// TwinCAT 3 PLC project nott_ics
// ProgramVersion: 3.1.4024.0
// libraries:
//   CmpBitmapPool, * (System)
//   ESO LDC Comm Common Library, * (ESO)
//   ESO LDC Comm Tcp Library, * (ESO)
//   ESO LDC Common Library, * (ESO)
//   ESO LDC Cryo Library, * (ESO)
//   ESO LDC Motor Library, * (ESO)
//   ESO LDC Shutter Library, * (ESO)
//   ESO LDC Timer Library, * (ESO)
//   Tc2_EtherCAT, * (Beckhoff Automation GmbH)
//   Tc2_MC2, * (Beckhoff Automation GmbH)
//   Tc2_Standard, * (Beckhoff Automation GmbH)
//   Tc2_System, * (Beckhoff Automation GmbH)
//   Tc2_Utilities, * (Beckhoff Automation GmbH)
//   Tc3_Module, * (Beckhoff Automation GmbH)
//   VisuDialogs, * (System)
// project tree:
//   / CameraTrigs.TcTTO, GlobalTextList.TcGTLO, PlcTask.TcTTO, Visualization Manager.TcVMO (not stored), VISU_TASK.TcTTO
//   DUTs/Structures/ T_NOTT_STAT.TcDUT
//   DUTs/ T_NOTT_IR_CAMERA_DL_SYNC.TcDUT, T_NOTT_CAMERA_TIMESTAMPS_N_DL_POS.TcDUT
//   GVLs/ NOTT_GVL.TcGVL
//   HMI/DUTs/Subsystems/Tip_Tilt/ E_HMI_TIP_TILT_TABS.TcDUT
//   HMI/DUTs/System/ E_HMI_TABS.TcDUT
//   HMI/DUTs/Util/ E_HMI_COLORS.TcDUT, E_HMI_VOTER_TABS.TcDUT, T_ECAT_MODULE.TcDUT, T_HMI_COLORS.TcDUT
//   HMI/POUs/Devices/Cabinets/ FB_HMI_CABINETS.TcPOU
//   HMI/POUs/Devices/Control_Loops/ FB_HMI_CONTROL_LOOPS.TcPOU, FB_HMI_METIS_CTRL_TEMPERATURE.TcPOU
//   HMI/POUs/Devices/Control_Units/ FB_HMI_CONTROL_UNITS.TcPOU
//   HMI/POUs/Devices/Coolers/ FB_HMI_COOLERS.TcPOU
//   HMI/POUs/Devices/Detectors/ FB_HMI_DETECTORS.TcPOU
//   HMI/POUs/Devices/Heaters/ FB_HMI_HEATERS.TcPOU, FB_HMI_METIS_HEATER.TcPOU
//   HMI/POUs/Devices/Lakeshores/ FB_HMI_LAKESHORE.TcPOU
//   HMI/POUs/Devices/Pressures/ FB_HMI_PRESSURES.TcPOU
//   HMI/POUs/Devices/Pumps/ FB_HMI_PUMPS.TcPOU, FB_HMI_RP_BRANCH_A.TcPOU, FB_HMI_RP_BRANCH_B.TcPOU, FB_HMI_TP_BRANCH_A.TcPOU, FB_HMI_TP_BRANCH_B.TcPOU
//   HMI/POUs/Devices/RH/ FB_HMI_METIS_RH_SENSOR.TcPOU
//   HMI/POUs/Devices/Temperatures/Components/ FB_HMI_TEMP_VOTERS.TcPOU
//   HMI/POUs/Devices/Temperatures/ FB_HMI_TEMPERATURES.TcPOU
//   HMI/POUs/Devices/Valves/ FB_HMI_VALVES.TcPOU
//   HMI/POUs/Devices/Voters/ FB_HMI_VOTER.TcPOU
//   HMI/POUs/Events/ FB_HMI_EVENTS.TcPOU
//   HMI/POUs/CRYO_Interlocks/ FB_HMI_CRYO_INTERLOCKS.TcPOU
//   HMI/POUs/Services/ FB_HMI_SERVICES.TcPOU, FB_HMI_SERVICES_TIME.TcPOU
//   HMI/POUs/Services/Status/ FB_HMI_BUSY_STATUS.TcPOU, FB_HMI_HEALTH_STATUS.TcPOU, FB_HMI_STATUS.TcPOU, F_HMI_BUSY_TO_COLOR.TcPOU, F_HMI_HEALTH_BUSY_TO_COLOR.TcPOU, F_HMI_HEALTH_TO_COLOR.TcPOU
//   HMI/POUs/Subsystems/Beam_Splitter/ FB_HMI_CALIBRATION_BEAM_SPLITTER.TcPOU
//   HMI/POUs/Subsystems/Birefringence/ FB_HMI_BIREFRINGENCE.TcPOU
//   HMI/POUs/Subsystems/CO2_Pressure/ FB_HMI_CO2_PRESSURE_CONTROL.TcPOU
//   HMI/POUs/Subsystems/CO2_Translation_Stages/ FB_HMI_CO2_TRANS_STAGES.TcPOU
//   HMI/POUs/Subsystems/DelayLines/ FB_HMI_DELAY_LINES.TcPOU
//   HMI/POUs/Subsystems/Shutters/ FB_HMI_SHUTTERS.TcPOU
//   HMI/POUs/Subsystems/TipTilt/Components/ FB_HMI_TILT_A.TcPOU, FB_HMI_TILT_B.TcPOU, FB_HMI_TIP_A.TcPOU, FB_HMI_TIP_B.TcPOU
//   HMI/POUs/Subsystems/TipTilt/ FB_HMI_TIP_TILT.TcPOU
//   HMI/POUs/Subsystems/ZnSe_Actuators/ FB_HMI_ZNSE_ACTUATORS.TcPOU
//   HMI/POUs/Util/Button/ FB_HMI_BUTTON.TcPOU
//   HMI/POUs/Util/Component/ FB_HMI_COMPONENT.TcPOU
//   HMI/POUs/Util/Functions/ F_GetConnectionColor.TcPOU, F_GetConnectionString.TcPOU
//   HMI/ PRG_HMI.TcPOU, VISU_HMI.TcVIS
//   HMI/VISUs/Events/ VISU_HMI_EVENTS.TcVIS
//   HMI/VISUs/Home/ VISU_HMI_HOME.TcVIS
//   HMI/VISUs/ICS_Interlocks/ VISU_HMI_CRYO_INTERLOCKS.TcVIS
//   HMI/VISUs/Services/ VISU_HMI_SERVICES.TcVIS, VISU_HMI_SERVICES_TIME.TcVIS
//   HMI/VISUs/Subsystems/Beam_Splitter/ VISU_HMI_BEAM_SPLITTER.TcVIS
//   HMI/VISUs/Subsystems/Birefringence/ VISU_HMI_BIREFRINGENCE.TcVIS
//   HMI/VISUs/Subsystems/CO2_Pressure/ VISU_HMI_CO2_PRESSURE.TcVIS
//   HMI/VISUs/Subsystems/CO2_Translation_Stages/ VISU_HMI_CO2_TRANS_STAGES.TcVIS
//   HMI/VISUs/Subsystems/DelayLines/ VISU_HMI_DELAY_LINES.TcVIS
//   HMI/VISUs/Subsystems/Shutters/ VISU_HMI_SHUTTERS.TcVIS
//   HMI/VISUs/Subsystems/TipTilt/Components/ VISU_HMI_TILT_A.TcVIS, VISU_HMI_TILT_B.TcVIS, VISU_HMI_TIP_A.TcVIS, VISU_HMI_TIP_B.TcVIS
//   HMI/VISUs/Subsystems/TipTilt/ VISU_HMI_TIP_TILT.TcVIS
//   HMI/VISUs/Subsystems/ZnSe_Actuators/ VISU_HMI_ZNSE_ACTUATORS.TcVIS
//   HMI/VISUs/Templates/CO2_Valve/ GUI_TEMPLATE_ACTUATOR_ENG.TcVIS
//   HMI/VISUs/Templates/Motors/ GUI_TEMPLATE_MOTOR.TcVIS, GUI_TEMPLATE_NOTT_MOTOR_CONFIG.TcVIS, GUI_TEMPLATE_NOTT_MOTOR_CONTROL.TcVIS
//   HMI/VISUs/Templates/ NOTT_Images.TcIPO (not stored)
//   HMI/VISUs/Templates/Shutters/ GUI_TEMPLATE_NOTT_SHUTTER.TcVIS, GUI_TEMPLATE_SHUTTER_CONTROL.TcVIS
//   HMI/VISUs/Util/Button/ VISU_HMI_BUTTON_IMAGES.TcIPO (not stored), VISU_HMI_ROUTINES_BUTTON.TcVIS, VISU_HMI_SUBSUBSYSTEM_BUTTON.TcVIS, VISU_HMI_SUBSYSTEM_BUTTON.TcVIS, VISU_HMI_SYSTEM_BUTTON.TcVIS
//   HMI/VISUs/Util/ ICONS_IMAGE_POOL.TcIPO (not stored)
//   POUs/Camera_Triggers/ INFRATEC_TRIGERS.TcPOU
//   POUs/Cryo_Interlocks/ FB_NOTT_CRYO_INTERLOCKS.TcPOU
//   POUs/Devices/NOTT_Motor/ FB_NOTT_MOTOR.TcPOU
//   POUs/EVENTS/ FB_NOTT_EVENTS.TcPOU
//   POUs/Functions/ F_SysTimeToString.TcPOU
//   POUs/ MAIN.TcPOU
//   POUs/Services/ FB_SERVICES.TcPOU
//   POUs/Subsystems/ FB_NOTT_CO2_PRESSURE_CONTROL.TcPOU, FB_NOTT_CALIBRATION_BEAM_SPLITTER.TcPOU, FB_NOTT_ZNSE_ACTUATORS.TcPOU, FB_NOTT_DELAY_LINES.TcPOU, FB_NOTT_SHUTTERS.TcPOU, FB_NOTT_CO2_TRANS_STAGES.TcPOU, FB_NOTT_TIP_TILT.TcPOU, FB_NOTT_BIREFRINGENCE.TcPOU
//   POUs/System/ FB_NOTT_CRYO_CTRL.TcPOU, FB_NOTT_ICS.TcPOU
//   POUs/Valve/ FB_CRYO_BIN_CTRL.TcPOU, FB_CRYO_VALVE_CTRL.TcPOU
//   VISUs/GUIs/Cryo/ GUI_CRYO_TEMPS.TcVIS
//   VISUs/GUIs/NBS/ GUI_NOTT_NBS.TcVIS
//   VISUs/GUIs/Shutters/ GUI_TEST_STEPPER_SHUTTER.TcVIS, GUI_NOTT_SHUTTERS.TcVIS
//   VISUs/GUIs/Templates/ TEMPLATE_NOTT_CRYO_TEMPS.TcVIS
//   VISUs/GUIs/Delay_Lines/ GUI_NOTT_DL_CONFIG.TcVIS, GUI_NOTT_DL_CTRL.TcVIS
//   VISUs/GUIs/ GUI_NOTT_DL_1.TcVIS
//   VISUs/GUIs/Time/ GUI_NOTT_TIME.TcVIS
//   VISUs/GUIs/TipTilt/ GUI_NOTT_TIP_A_CONFIG.TcVIS, GUI_NOTT_TIP_B_CONFIG.TcVIS, GUI_NOTT_TILT_B_CONFIG.TcVIS, GUI_NOTT_TILT_A_CONFIG.TcVIS, GUI_NOTT_TIP_A_CTRL.TcVIS, GUI_NOTT_TIP_B_CTRL.TcVIS, GUI_NOTT_TILT_A_CTRL.TcVIS, GUI_NOTT_TILT_B_CTRL.TcVIS
//   VISUs/Templates/ MOTOR_CONTROL.TcVIS
// real-time tasks:
//   TASK PlcTask: cycle T#10ms, priority 20, ADS port 350
//   TASK CameraTrigs: cycle T#1ms, priority 1, ADS port 351
//   TASK VISU_TASK: cycle T#200000us, priority 30, ADS port 352
// motion (NC):
//   TASK NC-Task 1 SAF: cycle T#2ms, priority 4, ADS port 501
//   TASK NC-Task 1 SVB: cycle T#10ms, priority 8, ADS port 511
//   AXIS NTPA1 (id 23)
//     Dynamic: AccelerationMaximum=1.8, DecelerationMaximum=1.8, Acceleration=0.2525, Deceleration=0.2525, Jerk=15.9390625
//     Velo: RefSearch=0.05, RefSync=0.05, SlowManual=0.05, FastManual=0.1, Fast=0.4, Maximum=0.4
//     OtherSettings: AllowMotionCmdToSlave=true, PulseDistancePos=0.05, PulseDistanceNeg=0.05
//     encoder EncType=4
//       EncPara: ScaleFactorNumerator=3.05e-05, MaxCount=#x0000ffff
//         Inc: RefSoftSyncMask=#x0000ffff
//     drive DrvType=23
//       Analog: VeloReferenz=0.4, TorqueSetpointScale=10, ScaleFactorActTorque=0.1
//       TimeComp: TaskDelayCycles=1
//     controller CtrType=13
//       CtrPara: PriorControlFactor=1
//         PID: PosKp=50, PosTn=5, PosTd=0.5, DeadBandPosition=1e-05
//         Observer: ObserverMode=1, MotorTorqueConstant=2, BandWidth=20
//   AXIS NTPA2 (id 24)
//     Dynamic: AccelerationMaximum=1.8, DecelerationMaximum=1.8, Acceleration=0.2525, Deceleration=0.2525, Jerk=15.9390625
//     Velo: RefSearch=0.05, RefSync=0.05, SlowManual=0.05, FastManual=0.1, Fast=0.4, Maximum=0.4
//     OtherSettings: AllowMotionCmdToSlave=true, PulseDistancePos=0.05, PulseDistanceNeg=0.05
//     encoder EncType=4
//       EncPara: ScaleFactorNumerator=3.05e-05, MaxCount=#x0000ffff
//         Inc: RefSoftSyncMask=#x0000ffff
//     drive DrvType=23
//       Analog: VeloReferenz=0.4, TorqueSetpointScale=10, ScaleFactorActTorque=0.1
//       TimeComp: TaskDelayCycles=1
//     controller CtrType=13
//       CtrPara: PriorControlFactor=1
//         PID: PosKp=50, PosTn=5, PosTd=0.5, DeadBandPosition=1e-05
//         Observer: ObserverMode=1, MotorTorqueConstant=2, BandWidth=20
//   AXIS NTPA3 (id 25)
//     Dynamic: AccelerationMaximum=1.8, DecelerationMaximum=1.8, Acceleration=0.2525, Deceleration=0.2525, Jerk=15.9390625
//     Velo: RefSearch=0.05, RefSync=0.05, SlowManual=0.05, FastManual=0.1, Fast=0.4, Maximum=0.4
//     OtherSettings: AllowMotionCmdToSlave=true, PulseDistancePos=0.05, PulseDistanceNeg=0.05
//     encoder EncType=4
//       EncPara: ScaleFactorNumerator=3.05e-05, MaxCount=#x0000ffff
//         Inc: RefSoftSyncMask=#x0000ffff
//     drive DrvType=23
//       Analog: VeloReferenz=0.4, TorqueSetpointScale=10, ScaleFactorActTorque=0.1
//       TimeComp: TaskDelayCycles=1
//     controller CtrType=13
//       CtrPara: PriorControlFactor=1
//         PID: PosKp=50, PosTn=5, PosTd=0.5, DeadBandPosition=1e-05
//         Observer: ObserverMode=1, MotorTorqueConstant=2, BandWidth=20
//   AXIS NTPA4 (id 26)
//     Dynamic: AccelerationMaximum=1.8, DecelerationMaximum=1.8, Acceleration=0.2525, Deceleration=0.2525, Jerk=15.9390625
//     Velo: RefSearch=0.05, RefSync=0.05, SlowManual=0.05, FastManual=0.1, Fast=0.4, Maximum=0.4
//     OtherSettings: AllowMotionCmdToSlave=true, PulseDistancePos=0.05, PulseDistanceNeg=0.05
//     encoder EncType=4
//       EncPara: ScaleFactorNumerator=3.05e-05, MaxCount=#x0000ffff
//         Inc: RefSoftSyncMask=#x0000ffff
//     drive DrvType=23
//       Analog: VeloReferenz=0.4, TorqueSetpointScale=10, ScaleFactorActTorque=0.1
//       TimeComp: TaskDelayCycles=1
//     controller CtrType=13
//       CtrPara: PriorControlFactor=1
//         PID: PosKp=50, PosTn=5, PosTd=0.5, DeadBandPosition=1e-05
//         Observer: ObserverMode=1, MotorTorqueConstant=2, BandWidth=20
//   AXIS NTTA1 (id 27)
//     Dynamic: AccelerationMaximum=1.8, DecelerationMaximum=1.8, Acceleration=0.2525, Deceleration=0.2525, Jerk=15.9390625
//     Velo: RefSearch=0.05, RefSync=0.05, SlowManual=0.05, FastManual=0.1, Fast=0.4, Maximum=0.4
//     OtherSettings: AllowMotionCmdToSlave=true, PulseDistancePos=0.05, PulseDistanceNeg=0.05
//     encoder EncType=4
//       EncPara: ScaleFactorNumerator=3.05e-05, MaxCount=#x0000ffff
//         Inc: RefSoftSyncMask=#x0000ffff
//     drive DrvType=23
//       Analog: VeloReferenz=0.4, TorqueSetpointScale=10, ScaleFactorActTorque=0.1
//       TimeComp: TaskDelayCycles=1
//     controller CtrType=13
//       CtrPara: PriorControlFactor=1
//         PID: PosKp=50, PosTn=5, PosTd=0.5, DeadBandPosition=1e-05
//         Observer: ObserverMode=1, MotorTorqueConstant=2, BandWidth=20
//   AXIS NTTA2 (id 28)
//     Dynamic: AccelerationMaximum=1.8, DecelerationMaximum=1.8, Acceleration=0.2525, Deceleration=0.2525, Jerk=15.9390625
//     Velo: RefSearch=0.05, RefSync=0.05, SlowManual=0.05, FastManual=0.1, Fast=0.4, Maximum=0.4
//     OtherSettings: AllowMotionCmdToSlave=true, PulseDistancePos=0.05, PulseDistanceNeg=0.05
//     encoder EncType=4
//       EncPara: ScaleFactorNumerator=3.05e-05, MaxCount=#x0000ffff
//         Inc: RefSoftSyncMask=#x0000ffff
//     drive DrvType=23
//       Analog: VeloReferenz=0.4, TorqueSetpointScale=10, ScaleFactorActTorque=0.1
//       TimeComp: TaskDelayCycles=1
//     controller CtrType=13
//       CtrPara: PriorControlFactor=1
//         PID: PosKp=50, PosTn=5, PosTd=0.5, DeadBandPosition=1e-05
//         Observer: ObserverMode=1, MotorTorqueConstant=2, BandWidth=20
//   AXIS NTTA3 (id 29)
//     Dynamic: AccelerationMaximum=1.8, DecelerationMaximum=1.8, Acceleration=0.2525, Deceleration=0.2525, Jerk=15.9390625
//     Velo: RefSearch=0.05, RefSync=0.05, SlowManual=0.05, FastManual=0.1, Fast=0.4, Maximum=0.4
//     OtherSettings: AllowMotionCmdToSlave=true, PulseDistancePos=0.05, PulseDistanceNeg=0.05
//     encoder EncType=4
//       EncPara: ScaleFactorNumerator=3.05e-05, MaxCount=#x0000ffff
//         Inc: RefSoftSyncMask=#x0000ffff
//     drive DrvType=23
//       Analog: VeloReferenz=0.4, TorqueSetpointScale=10, ScaleFactorActTorque=0.1
//       TimeComp: TaskDelayCycles=1
//     controller CtrType=13
//       CtrPara: PriorControlFactor=1
//         PID: PosKp=50, PosTn=5, PosTd=0.5, DeadBandPosition=1e-05
//         Observer: ObserverMode=1, MotorTorqueConstant=2, BandWidth=20
//   AXIS NTTA4 (id 30)
//     Dynamic: AccelerationMaximum=1.8, DecelerationMaximum=1.8, Acceleration=0.2525, Deceleration=0.2525, Jerk=15.9390625
//     Velo: RefSearch=0.05, RefSync=0.05, SlowManual=0.05, FastManual=0.1, Fast=0.4, Maximum=0.4
//     OtherSettings: AllowMotionCmdToSlave=true, PulseDistancePos=0.05, PulseDistanceNeg=0.05
//     encoder EncType=4
//       EncPara: ScaleFactorNumerator=3.05e-05, MaxCount=#x0000ffff
//         Inc: RefSoftSyncMask=#x0000ffff
//     drive DrvType=23
//       Analog: VeloReferenz=0.4, TorqueSetpointScale=10, ScaleFactorActTorque=0.1
//       TimeComp: TaskDelayCycles=1
//     controller CtrType=13
//       CtrPara: PriorControlFactor=1
//         PID: PosKp=50, PosTn=5, PosTd=0.5, DeadBandPosition=1e-05
//         Observer: ObserverMode=1, MotorTorqueConstant=2, BandWidth=20
//   AXIS NTPB1 (id 31)
//     Dynamic: AccelerationMaximum=1.8, DecelerationMaximum=1.8, Acceleration=0.2525, Deceleration=0.2525, Jerk=15.9390625
//     Velo: RefSearch=0.05, RefSync=0.05, SlowManual=0.05, FastManual=0.1, Fast=0.4, Maximum=0.4
//     OtherSettings: AllowMotionCmdToSlave=true, PulseDistancePos=0.05, PulseDistanceNeg=0.05
//     encoder EncType=4
//       EncPara: ScaleFactorNumerator=3.05e-05, MaxCount=#x0000ffff
//         Inc: RefSoftSyncMask=#x0000ffff
//     drive DrvType=23
//       Analog: VeloReferenz=0.4, TorqueSetpointScale=10, ScaleFactorActTorque=0.1
//       TimeComp: TaskDelayCycles=1
//     controller CtrType=13
//       CtrPara: PriorControlFactor=1
//         PID: PosKp=50, PosTn=5, PosTd=0.5, DeadBandPosition=1e-05
//         Observer: ObserverMode=1, MotorTorqueConstant=2, BandWidth=20
//   AXIS NTPB2 (id 32)
//     Dynamic: AccelerationMaximum=1.8, DecelerationMaximum=1.8, Acceleration=0.2525, Deceleration=0.2525, Jerk=15.9390625
//     Velo: RefSearch=0.05, RefSync=0.05, SlowManual=0.05, FastManual=0.1, Fast=0.4, Maximum=0.4
//     OtherSettings: AllowMotionCmdToSlave=true, PulseDistancePos=0.05, PulseDistanceNeg=0.05
//     encoder EncType=4
//       EncPara: ScaleFactorNumerator=3.05e-05, MaxCount=#x0000ffff
//         Inc: RefSoftSyncMask=#x0000ffff
//     drive DrvType=23
//       Analog: VeloReferenz=0.4, TorqueSetpointScale=10, ScaleFactorActTorque=0.1
//       TimeComp: TaskDelayCycles=1
//     controller CtrType=13
//       CtrPara: PriorControlFactor=1
//         PID: PosKp=50, PosTn=5, PosTd=0.5, DeadBandPosition=1e-05
//         Observer: ObserverMode=1, MotorTorqueConstant=2, BandWidth=20
//   AXIS NTPB3 (id 33)
//     Dynamic: AccelerationMaximum=1.8, DecelerationMaximum=1.8, Acceleration=0.2525, Deceleration=0.2525, Jerk=15.9390625
//     Velo: RefSearch=0.05, RefSync=0.05, SlowManual=0.05, FastManual=0.1, Fast=0.4, Maximum=0.4
//     OtherSettings: AllowMotionCmdToSlave=true, PulseDistancePos=0.05, PulseDistanceNeg=0.05
//     encoder EncType=4
//       EncPara: ScaleFactorNumerator=3.05e-05, MaxCount=#x0000ffff
//         Inc: RefSoftSyncMask=#x0000ffff
//     drive DrvType=23
//       Analog: VeloReferenz=0.4, TorqueSetpointScale=10, ScaleFactorActTorque=0.1
//       TimeComp: TaskDelayCycles=1
//     controller CtrType=13
//       CtrPara: PriorControlFactor=1
//         PID: PosKp=50, PosTn=5, PosTd=0.5, DeadBandPosition=1e-05
//         Observer: ObserverMode=1, MotorTorqueConstant=2, BandWidth=20
//   AXIS NTPB4 (id 34)
//     Dynamic: AccelerationMaximum=1.8, DecelerationMaximum=1.8, Acceleration=0.2525, Deceleration=0.2525, Jerk=15.9390625
//     Velo: RefSearch=0.05, RefSync=0.05, SlowManual=0.05, FastManual=0.1, Fast=0.4, Maximum=0.4
//     OtherSettings: AllowMotionCmdToSlave=true, PulseDistancePos=0.05, PulseDistanceNeg=0.05
//     encoder EncType=4
//       EncPara: ScaleFactorNumerator=3.05e-05, MaxCount=#x0000ffff
//         Inc: RefSoftSyncMask=#x0000ffff
//     drive DrvType=23
//       Analog: VeloReferenz=0.4, TorqueSetpointScale=10, ScaleFactorActTorque=0.1
//       TimeComp: TaskDelayCycles=1
//     controller CtrType=13
//       CtrPara: PriorControlFactor=1
//         PID: PosKp=50, PosTn=5, PosTd=0.5, DeadBandPosition=1e-05
//         Observer: ObserverMode=1, MotorTorqueConstant=2, BandWidth=20
//   AXIS NTTB1 (id 36)
//     Dynamic: AccelerationMaximum=1.8, DecelerationMaximum=1.8, Acceleration=0.2525, Deceleration=0.2525, Jerk=15.9390625
//     Velo: RefSearch=0.05, RefSync=0.05, SlowManual=0.05, FastManual=0.1, Fast=0.4, Maximum=0.4
//     OtherSettings: AllowMotionCmdToSlave=true, PulseDistancePos=0.05, PulseDistanceNeg=0.05
//     encoder EncType=4
//       EncPara: ScaleFactorNumerator=3.05e-05, MaxCount=#x0000ffff
//         Inc: RefSoftSyncMask=#x0000ffff
//     drive DrvType=23
//       Analog: VeloReferenz=0.4, TorqueSetpointScale=10, ScaleFactorActTorque=0.1
//       TimeComp: TaskDelayCycles=1
//     controller CtrType=13
//       CtrPara: PriorControlFactor=1
//         PID: PosKp=50, PosTn=5, PosTd=0.5, DeadBandPosition=1e-05
//         Observer: ObserverMode=1, MotorTorqueConstant=2, BandWidth=20
//   AXIS NTTB2 (id 37)
//     Dynamic: AccelerationMaximum=1.8, DecelerationMaximum=1.8, Acceleration=0.2525, Deceleration=0.2525, Jerk=15.9390625
//     Velo: RefSearch=0.05, RefSync=0.05, SlowManual=0.05, FastManual=0.1, Fast=0.4, Maximum=0.4
//     OtherSettings: AllowMotionCmdToSlave=true, PulseDistancePos=0.05, PulseDistanceNeg=0.05
//     encoder EncType=4
//       EncPara: ScaleFactorNumerator=3.05e-05, MaxCount=#x0000ffff
//         Inc: RefSoftSyncMask=#x0000ffff
//     drive DrvType=23
//       Analog: VeloReferenz=0.4, TorqueSetpointScale=10, ScaleFactorActTorque=0.1
//       TimeComp: TaskDelayCycles=1
//     controller CtrType=13
//       CtrPara: PriorControlFactor=1
//         PID: PosKp=50, PosTn=5, PosTd=0.5, DeadBandPosition=1e-05
//         Observer: ObserverMode=1, MotorTorqueConstant=2, BandWidth=20
//   AXIS NTTB3 (id 38)
//     Dynamic: AccelerationMaximum=1.8, DecelerationMaximum=1.8, Acceleration=0.2525, Deceleration=0.2525, Jerk=15.9390625
//     Velo: RefSearch=0.05, RefSync=0.05, SlowManual=0.05, FastManual=0.1, Fast=0.4, Maximum=0.4
//     OtherSettings: AllowMotionCmdToSlave=true, PulseDistancePos=0.05, PulseDistanceNeg=0.05
//     encoder EncType=4
//       EncPara: ScaleFactorNumerator=3.05e-05, MaxCount=#x0000ffff
//         Inc: RefSoftSyncMask=#x0000ffff
//     drive DrvType=23
//       Analog: VeloReferenz=0.4, TorqueSetpointScale=10, ScaleFactorActTorque=0.1
//       TimeComp: TaskDelayCycles=1
//     controller CtrType=13
//       CtrPara: PriorControlFactor=1
//         PID: PosKp=50, PosTn=5, PosTd=0.5, DeadBandPosition=1e-05
//         Observer: ObserverMode=1, MotorTorqueConstant=2, BandWidth=20
//   AXIS NTTB4 (id 39)
//     Dynamic: AccelerationMaximum=1.8, DecelerationMaximum=1.8, Acceleration=0.2525, Deceleration=0.2525, Jerk=15.9390625
//     Velo: RefSearch=0.05, RefSync=0.05, SlowManual=0.05, FastManual=0.1, Fast=0.4, Maximum=0.4
//     OtherSettings: AllowMotionCmdToSlave=true, PulseDistancePos=0.05, PulseDistanceNeg=0.05
//     encoder EncType=4
//       EncPara: ScaleFactorNumerator=3.05e-05, MaxCount=#x0000ffff
//         Inc: RefSoftSyncMask=#x0000ffff
//     drive DrvType=23
//       Analog: VeloReferenz=0.4, TorqueSetpointScale=10, ScaleFactorActTorque=0.1
//       TimeComp: TaskDelayCycles=1
//     controller CtrType=13
//       CtrPara: PriorControlFactor=1
//         PID: PosKp=50, PosTn=5, PosTd=0.5, DeadBandPosition=1e-05
//         Observer: ObserverMode=1, MotorTorqueConstant=2, BandWidth=20
//   AXIS NDL1 (id 19)
//     Dynamic: AccelerationMaximum=0.3, DecelerationMaximum=0.3, Acceleration=0.3, Deceleration=0.3, Jerk=0.5
//     Velo: RefSearch=0.05, RefSync=0.05, SlowManual=0.02, FastManual=0.075, Fast=0.2, Maximum=0.2
//     OtherSettings: AllowMotionCmdToSlave=true, PulseDistancePos=0.02, PulseDistanceNeg=0.02
//     encoder EncType=4
//       EncPara: ScaleFactorNumerator=1.5259e-06, MaxCount=#x0000ffff
//         Inc: RefSoftSyncMask=#x0000ffff
//     drive DrvType=24
//       Analog: VeloReferenz=0.2, TorqueSetpointScale=10, ScaleFactorActTorque=0.1
//       TimeComp: TaskDelayCycles=1
//     controller CtrType=1
//       CtrPara: PriorControlFactor=1
//         Observer: BandWidth=20
//   AXIS NDL2 (id 20)
//     Dynamic: AccelerationMaximum=0.3, DecelerationMaximum=0.3, Acceleration=0.3, Deceleration=0.3, Jerk=0.5
//     Velo: RefSearch=0.05, RefSync=0.05, SlowManual=0.02, FastManual=0.075, Fast=0.2, Maximum=0.2
//     OtherSettings: AllowMotionCmdToSlave=true, PulseDistancePos=0.02, PulseDistanceNeg=0.02
//     encoder EncType=4
//       EncPara: ScaleFactorNumerator=1.5259e-06, MaxCount=#x0000ffff
//         Inc: RefSoftSyncMask=#x0000ffff
//     drive DrvType=24
//       Analog: VeloReferenz=0.2, TorqueSetpointScale=10, ScaleFactorActTorque=0.1
//       TimeComp: TaskDelayCycles=1
//     controller CtrType=1
//       CtrPara: PriorControlFactor=1
//         Observer: BandWidth=20
//   AXIS NDL3 (id 21)
//     Dynamic: AccelerationMaximum=0.3, DecelerationMaximum=0.3, Acceleration=0.3, Deceleration=0.3, Jerk=0.5
//     Velo: RefSearch=0.05, RefSync=0.05, SlowManual=0.02, FastManual=0.075, Fast=0.2, Maximum=0.2
//     OtherSettings: AllowMotionCmdToSlave=true, PulseDistancePos=0.02, PulseDistanceNeg=0.02
//     encoder EncType=4
//       EncPara: ScaleFactorNumerator=1.5259e-06, MaxCount=#x0000ffff
//         Inc: RefSoftSyncMask=#x0000ffff
//     drive DrvType=24
//       Analog: VeloReferenz=0.2, TorqueSetpointScale=10, ScaleFactorActTorque=0.1
//       TimeComp: TaskDelayCycles=1
//     controller CtrType=1
//       CtrPara: PriorControlFactor=1
//         Observer: BandWidth=20
//   AXIS NDL4 (id 22)
//     Dynamic: AccelerationMaximum=0.3, DecelerationMaximum=0.3, Acceleration=0.3, Deceleration=0.3, Jerk=0.5
//     Velo: RefSearch=0.05, RefSync=0.05, SlowManual=0.02, FastManual=0.075, Fast=0.2, Maximum=0.2
//     OtherSettings: AllowMotionCmdToSlave=true, PulseDistancePos=0.02, PulseDistanceNeg=0.02
//     encoder EncType=4
//       EncPara: ScaleFactorNumerator=1.5259e-06, MaxCount=#x0000ffff
//         Inc: RefSoftSyncMask=#x0000ffff
//     drive DrvType=24
//       Analog: VeloReferenz=0.2, TorqueSetpointScale=10, ScaleFactorActTorque=0.1
//       TimeComp: TaskDelayCycles=1
//     controller CtrType=1
//       CtrPara: PriorControlFactor=1
//         Observer: BandWidth=20
//   AXIS NSH1 (id 35)
//     Dynamic: AccelerationMaximum=100, DecelerationMaximum=100, Acceleration=9, Deceleration=9, Jerk=1000
//     Velo: RefSearch=3, RefSync=3, SlowManual=3, FastManual=5, Fast=30, Maximum=35
//     PositionAreaControl: Enable=false
//     OtherSettings: AllowMotionCmdToSlave=true, PulseDistancePos=1, PulseDistanceNeg=1
//     encoder EncType=4
//       EncPara: ScaleFactorNumerator=0.00234375, MaxCount=#x0000ffff
//         Inc: RefSoftSyncMask=#x0000ffff
//     drive DrvType=24
//       Analog: VeloReferenz=35, TorqueSetpointScale=10, ScaleFactorActTorque=0.1
//       TimeComp: TaskDelayCycles=1
//     controller CtrType=1
//       CtrPara: PriorControlFactor=1
//         PosDiffControl: Enable=false
//         PID: PosKp=10
//         Observer: BandWidth=20
//   AXIS NSH2 (id 16)
//     Dynamic: AccelerationMaximum=100, DecelerationMaximum=100, Acceleration=9, Deceleration=9, Jerk=1000
//     Velo: RefSearch=3, RefSync=3, SlowManual=3, FastManual=5, Fast=30, Maximum=35
//     PositionAreaControl: Enable=false
//     OtherSettings: AllowMotionCmdToSlave=true, PulseDistancePos=1, PulseDistanceNeg=1
//     encoder EncType=4
//       EncPara: ScaleFactorNumerator=0.00234375, MaxCount=#x0000ffff
//         Inc: RefSoftSyncMask=#x0000ffff
//     drive DrvType=24
//       Analog: VeloReferenz=35, TorqueSetpointScale=10, ScaleFactorActTorque=0.1
//       TimeComp: TaskDelayCycles=1
//     controller CtrType=1
//       CtrPara: PriorControlFactor=1
//         PosDiffControl: Enable=false
//         PID: PosKp=10
//         Observer: BandWidth=20
//   AXIS NSH3 (id 17)
//     Dynamic: AccelerationMaximum=100, DecelerationMaximum=100, Acceleration=9, Deceleration=9, Jerk=1000
//     Velo: RefSearch=3, RefSync=3, SlowManual=3, FastManual=5, Fast=30, Maximum=35
//     PositionAreaControl: Enable=false
//     OtherSettings: AllowMotionCmdToSlave=true, PulseDistancePos=1, PulseDistanceNeg=1
//     encoder EncType=4
//       EncPara: ScaleFactorNumerator=0.00234375, MaxCount=#x0000ffff
//         Inc: RefSoftSyncMask=#x0000ffff
//     drive DrvType=24
//       Analog: VeloReferenz=35, TorqueSetpointScale=10, ScaleFactorActTorque=0.1
//       TimeComp: TaskDelayCycles=1
//     controller CtrType=1
//       CtrPara: PriorControlFactor=1
//         PosDiffControl: Enable=false
//         PID: PosKp=10
//         Observer: BandWidth=20
//   AXIS NSH4 (id 18)
//     Dynamic: AccelerationMaximum=200, DecelerationMaximum=200, Acceleration=9, Deceleration=9, Jerk=726.357
//     Velo: RefSearch=3, RefSync=3, SlowManual=3, FastManual=5, Fast=30, Maximum=35
//     PositionAreaControl: Enable=false
//     OtherSettings: AllowMotionCmdToSlave=true, PulseDistancePos=1, PulseDistanceNeg=1
//     encoder EncType=4
//       EncPara: ScaleFactorNumerator=0.00234375, MaxCount=#x0000ffff
//         Inc: RefSoftSyncMask=#x0000ffff
//     drive DrvType=24
//       Analog: VeloReferenz=35, TorqueSetpointScale=10, ScaleFactorActTorque=0.1
//       TimeComp: TaskDelayCycles=1
//     controller CtrType=1
//       CtrPara: PriorControlFactor=1
//         PosDiffControl: Enable=false
//         PID: PosKp=10
//         Observer: BandWidth=20
//   AXIS NCP1 (id 1)
//     Dynamic: AccelerationMaximum=4.5, DecelerationMaximum=4.5, Acceleration=4.5, Deceleration=4.5, Jerk=9
//     Velo: RefSearch=0.5, RefSync=0.5, SlowManual=0.05, FastManual=0.05, Fast=2, Maximum=2.3
//     OtherSettings: AllowMotionCmdToSlave=true, PulseDistancePos=0.02, PulseDistanceNeg=0.02
//     encoder EncType=4
//       EncPara: ScaleFactorNumerator=2.893937e-05, MaxCount=#x0000ffff
//         Inc: RefSoftSyncMask=#x0000ffff
//     drive DrvType=23
//       Analog: VeloReferenz=2.3, TorqueSetpointScale=10, ScaleFactorActTorque=0.1
//       TimeComp: TaskDelayCycles=1
//     controller CtrType=1
//       CtrPara: PriorControlFactor=1
//         Observer: BandWidth=20
//   AXIS NCP2 (id 2)
//     Dynamic: AccelerationMaximum=4.5, DecelerationMaximum=4.5, Acceleration=4.5, Deceleration=4.5, Jerk=9
//     Velo: RefSearch=0.5, RefSync=0.5, SlowManual=0.05, FastManual=0.05, Fast=2, Maximum=2.3
//     OtherSettings: AllowMotionCmdToSlave=true, PulseDistancePos=0.02, PulseDistanceNeg=0.02
//     encoder EncType=4
//       EncPara: ScaleFactorNumerator=2.893937e-05, MaxCount=#x0000ffff
//         Inc: RefSoftSyncMask=#x0000ffff
//     drive DrvType=23
//       Analog: VeloReferenz=2.3, TorqueSetpointScale=10, ScaleFactorActTorque=0.1
//       TimeComp: TaskDelayCycles=1
//     controller CtrType=1
//       CtrPara: PriorControlFactor=1
//         Observer: BandWidth=20
//   AXIS NCP3 (id 3)
//     Dynamic: AccelerationMaximum=4.5, DecelerationMaximum=4.5, Acceleration=4.5, Deceleration=4.5, Jerk=9
//     Velo: RefSearch=0.5, RefSync=0.5, SlowManual=0.05, FastManual=0.05, Fast=2, Maximum=2.3
//     OtherSettings: AllowMotionCmdToSlave=true, PulseDistancePos=0.02, PulseDistanceNeg=0.02
//     encoder EncType=4
//       EncPara: ScaleFactorNumerator=2.893937e-05, MaxCount=#x0000ffff
//         Inc: RefSoftSyncMask=#x0000ffff
//     drive DrvType=23
//       Analog: VeloReferenz=2.3, TorqueSetpointScale=10, ScaleFactorActTorque=0.1
//       TimeComp: TaskDelayCycles=1
//     controller CtrType=1
//       CtrPara: PriorControlFactor=1
//         Observer: BandWidth=20
//   AXIS NCP4 (id 4)
//     Dynamic: AccelerationMaximum=4.5, DecelerationMaximum=4.5, Acceleration=4.5, Deceleration=4.5, Jerk=9
//     Velo: RefSearch=0.5, RefSync=0.5, SlowManual=0.05, FastManual=0.05, Fast=2, Maximum=2.3
//     OtherSettings: AllowMotionCmdToSlave=true, PulseDistancePos=0.02, PulseDistanceNeg=0.02
//     encoder EncType=4
//       EncPara: ScaleFactorNumerator=2.893937e-05, MaxCount=#x0000ffff
//         Inc: RefSoftSyncMask=#x0000ffff
//     drive DrvType=23
//       Analog: VeloReferenz=2.3, TorqueSetpointScale=10, ScaleFactorActTorque=0.1
//       TimeComp: TaskDelayCycles=1
//     controller CtrType=1
//       CtrPara: PriorControlFactor=1
//         Observer: BandWidth=20
//   AXIS NGP1 (id 5)
//     Dynamic: AccelerationMaximum=4.5, DecelerationMaximum=4.5, Acceleration=4.5, Deceleration=4.5, Jerk=9
//     Velo: RefSearch=0.5, RefSync=0.5, SlowManual=0.05, FastManual=0.05, Fast=2, Maximum=2.3
//     OtherSettings: AllowMotionCmdToSlave=true, PulseDistancePos=0.02, PulseDistanceNeg=0.02
//     encoder EncType=4
//       EncPara: ScaleFactorNumerator=2.893937e-05, MaxCount=#x0000ffff
//         Inc: RefSoftSyncMask=#x0000ffff
//     drive DrvType=23
//       Analog: VeloReferenz=2.3, TorqueSetpointScale=10, ScaleFactorActTorque=0.1
//       TimeComp: TaskDelayCycles=1
//     controller CtrType=1
//       CtrPara: PriorControlFactor=1
//         Observer: BandWidth=20
//   AXIS NGP2 (id 6)
//     Dynamic: AccelerationMaximum=4.5, DecelerationMaximum=4.5, Acceleration=4.5, Deceleration=4.5, Jerk=9
//     Velo: RefSearch=0.5, RefSync=0.5, SlowManual=0.05, FastManual=0.05, Fast=2, Maximum=2.3
//     OtherSettings: AllowMotionCmdToSlave=true, PulseDistancePos=0.02, PulseDistanceNeg=0.02
//     encoder EncType=4
//       EncPara: ScaleFactorNumerator=2.893937e-05, MaxCount=#x0000ffff
//         Inc: RefSoftSyncMask=#x0000ffff
//     drive DrvType=23
//       Analog: VeloReferenz=2.3, TorqueSetpointScale=10, ScaleFactorActTorque=0.1
//       TimeComp: TaskDelayCycles=1
//     controller CtrType=1
//       CtrPara: PriorControlFactor=1
//         Observer: BandWidth=20
//   AXIS NGP3 (id 7)
//     Dynamic: AccelerationMaximum=4.5, DecelerationMaximum=4.5, Acceleration=4.5, Deceleration=4.5, Jerk=9
//     Velo: RefSearch=0.5, RefSync=0.5, SlowManual=0.05, FastManual=0.05, Fast=2, Maximum=2.3
//     OtherSettings: AllowMotionCmdToSlave=true, PulseDistancePos=0.02, PulseDistanceNeg=0.02
//     encoder EncType=4
//       EncPara: ScaleFactorNumerator=2.893937e-05, MaxCount=#x0000ffff
//         Inc: RefSoftSyncMask=#x0000ffff
//     drive DrvType=23
//       Analog: VeloReferenz=2.3, TorqueSetpointScale=10, ScaleFactorActTorque=0.1
//       TimeComp: TaskDelayCycles=1
//     controller CtrType=1
//       CtrPara: PriorControlFactor=1
//         Observer: BandWidth=20
//   AXIS NGP4 (id 8)
//     Dynamic: AccelerationMaximum=4.5, DecelerationMaximum=4.5, Acceleration=4.5, Deceleration=4.5, Jerk=9
//     Velo: RefSearch=0.5, RefSync=0.5, SlowManual=0.05, FastManual=0.05, Fast=2, Maximum=2.3
//     OtherSettings: AllowMotionCmdToSlave=true, PulseDistancePos=0.02, PulseDistanceNeg=0.02
//     encoder EncType=4
//       EncPara: ScaleFactorNumerator=2.893937e-05, MaxCount=#x0000ffff
//         Inc: RefSoftSyncMask=#x0000ffff
//     drive DrvType=23
//       Analog: VeloReferenz=2.3, TorqueSetpointScale=10, ScaleFactorActTorque=0.1
//       TimeComp: TaskDelayCycles=1
//     controller CtrType=1
//       CtrPara: PriorControlFactor=1
//         Observer: BandWidth=20
//   AXIS NBS (id 9)
//     Dynamic: AccelerationMaximum=4.5, DecelerationMaximum=4.5, Acceleration=4.5, Deceleration=4.5, Jerk=9
//     Velo: RefSearch=0.5, RefSync=0.5, SlowManual=0.05, FastManual=0.05, Fast=2, Maximum=2.3
//     OtherSettings: AllowMotionCmdToSlave=true, PulseDistancePos=0.02, PulseDistanceNeg=0.02
//     encoder EncType=4
//       EncPara: ScaleFactorNumerator=2.893937e-05, MaxCount=#x0000ffff
//         Inc: RefSoftSyncMask=#x0000ffff
//     drive DrvType=23
//       Analog: VeloReferenz=2.3, TorqueSetpointScale=10, ScaleFactorActTorque=0.1
//       TimeComp: TaskDelayCycles=1
//     controller CtrType=1
//       CtrPara: PriorControlFactor=1
//         Observer: BandWidth=20
//   AXIS NPC1 (id 11)
//     General: UnitName=Degree
//     Dynamic: AccelerationMaximum=4.5, DecelerationMaximum=4.5, Acceleration=4.5, Deceleration=4.5, Jerk=9
//     Velo: RefSearch=0.5, RefSync=0.5, SlowManual=0.05, FastManual=0.05, Fast=2, Maximum=25
//     OtherSettings: AllowMotionCmdToSlave=true, PulseDistancePos=0.02, PulseDistanceNeg=0.02
//     encoder EncType=4
//       EncPara: ScaleFactorNumerator=0.0005, MaxCount=#x0000ffff
//         Inc: RefSoftSyncMask=#x0000ffff
//     drive DrvType=23
//       Analog: VeloReferenz=25, TorqueSetpointScale=10, ScaleFactorActTorque=0.1
//       TimeComp: TaskDelayCycles=1
//     controller CtrType=1
//       CtrPara: PriorControlFactor=1
//         PID: PosKp=10
//         Observer: BandWidth=20
//   AXIS NPC2 (id 12)
//     Dynamic: AccelerationMaximum=4.5, DecelerationMaximum=4.5, Acceleration=4.5, Deceleration=4.5, Jerk=9
//     Velo: RefSearch=0.5, RefSync=0.5, SlowManual=0.05, FastManual=0.05, Fast=2, Maximum=2.3
//     OtherSettings: AllowMotionCmdToSlave=true, PulseDistancePos=0.02, PulseDistanceNeg=0.02
//     encoder EncType=4
//       EncPara: ScaleFactorNumerator=2.893937e-05, MaxCount=#x0000ffff
//         Inc: RefSoftSyncMask=#x0000ffff
//     drive DrvType=23
//       Analog: VeloReferenz=2.3, TorqueSetpointScale=10, ScaleFactorActTorque=0.1
//       TimeComp: TaskDelayCycles=1
//     controller CtrType=1
//       CtrPara: PriorControlFactor=1
//         Observer: BandWidth=20
//   AXIS NPC3 (id 13)
//     Dynamic: AccelerationMaximum=4.5, DecelerationMaximum=4.5, Acceleration=4.5, Deceleration=4.5, Jerk=9
//     Velo: RefSearch=0.5, RefSync=0.5, SlowManual=0.05, FastManual=0.05, Fast=2, Maximum=2.3
//     OtherSettings: AllowMotionCmdToSlave=true, PulseDistancePos=0.02, PulseDistanceNeg=0.02
//     encoder EncType=4
//       EncPara: ScaleFactorNumerator=2.893937e-05, MaxCount=#x0000ffff
//         Inc: RefSoftSyncMask=#x0000ffff
//     drive DrvType=23
//       Analog: VeloReferenz=2.3, TorqueSetpointScale=10, ScaleFactorActTorque=0.1
//       TimeComp: TaskDelayCycles=1
//     controller CtrType=1
//       CtrPara: PriorControlFactor=1
//         Observer: BandWidth=20
//   AXIS NPC4 (id 14)
//     Dynamic: AccelerationMaximum=4.5, DecelerationMaximum=4.5, Acceleration=4.5, Deceleration=4.5, Jerk=9
//     Velo: RefSearch=0.5, RefSync=0.5, SlowManual=0.05, FastManual=0.05, Fast=2, Maximum=2.3
//     OtherSettings: AllowMotionCmdToSlave=true, PulseDistancePos=0.02, PulseDistanceNeg=0.02
//     encoder EncType=4
//       EncPara: ScaleFactorNumerator=2.893937e-05, MaxCount=#x0000ffff
//         Inc: RefSoftSyncMask=#x0000ffff
//     drive DrvType=23
//       Analog: VeloReferenz=2.3, TorqueSetpointScale=10, ScaleFactorActTorque=0.1
//       TimeComp: TaskDelayCycles=1
//     controller CtrType=1
//       CtrPara: PriorControlFactor=1
//         Observer: BandWidth=20
// I/O:
//   DEVICE Device 6 (NOV-DP-RAM)
//   DEVICE Device 1 (EtherCAT), AmsNetId 5.134.125.93.2.1
//     Term 1 (EK1200) [EK1200-5000 EtherCAT Power supply (2A E-Bus)]
//       Term 2 (EL6070-0033) [EL6070-0033 1Ch. Licence key terminal, individual licences]
//       Term 3 (EL1008) [EL1008 8Ch. Dig. Input 24V, 3ms]
//       Term 4 (EL2008) [EL2008 8Ch. Dig. Output 24V, 0.5A]
//       Term 5 (EL6688) [EL6688 - External Synchronisation Interface (IEEE1588)]
//       Term 6 (EK1122) [EK1122 2 port EtherCAT junction]
//       Term 51 (EK1122) [EK1122 2 port EtherCAT junction]
//       Term 55 (EL9011) [EL9011 End Terminal]
//     Term 7 (EK1101) [EK1101 EtherCAT Coupler (2A E-Bus, ID switch)]
//       Term 8 (EL2004) [EL2004 4Ch. Dig. Output 24V, 0.5A]
//       Term 9 (EL3218) [EL3218-0000 8Ch. Ana. Input PT100 (RTD)]
//       Term 10 (EL9505) [EL9505 Power supply terminal 5V]
//       Term 11 (EL9505) [EL9505 Power supply terminal 5V]
//       Term 12 (EL9505) [EL9505 Power supply terminal 5V]
//       Term 13 (EL9505) [EL9505 Power supply terminal 5V]
//       Term 14 (EK1122) [EK1122 2 port EtherCAT junction]
//         Term 15 (EK1101) [EK1101 EtherCAT Coupler (2A E-Bus, ID switch)]
//           NCP1 - NCP2 (N1) (EL7342) [EL7342 2Ch. DC motor output stage (50V, 3.5A)]
//           NCP3 - NCP4 (N2) (EL7342) [EL7342 2Ch. DC motor output stage (50V, 3.5A)]
//           N3 (EL1008) [EL1008 8Ch. Dig. Input 24V, 3ms]
//           NGP1 - NGP2 (N5) (EL7342) [EL7342 2Ch. DC motor output stage (50V, 3.5A)]
//           NGP3 - NGP4 (N6) (EL7342) [EL7342 2Ch. DC motor output stage (50V, 3.5A)]
//           N7 (EL1008) [EL1008 8Ch. Dig. Input 24V, 3ms]
//           NBS (N8) (EL7342) [EL7342 2Ch. DC motor output stage (50V, 3.5A)]
//           N9 (EL1008) [EL1008 8Ch. Dig. Input 24V, 3ms]
//           NPC1 - NPC2 (N11) (EL7342) [EL7342 2Ch. DC motor output stage (50V, 3.5A)]
//           NPC3 - NPC4 (N12) (EL7342) [EL7342 2Ch. DC motor output stage (50V, 3.5A)]
//           N13 (EL1008) [EL1008 8Ch. Dig. Input 24V, 3ms]
//           Power (N14) (EL9410) [EL9410 E-Bus Power Supplier  (Diagnostics)]
//           NSH1 (N16) (EL7047) [EL7047 1Ch. Stepper motor output stage (50V, 5A)]
//           NSH2 (N17) (EL7047) [EL7047 1Ch. Stepper motor output stage (50V, 5A)]
//           NSH3 (N18) (EL7047) [EL7047 1Ch. Stepper motor output stage (50V, 5A)]
//           NSH4 (N19) (EL7047) [EL7047 1Ch. Stepper motor output stage (50V, 5A)]
//           Term 52 (EL9011) [EL9011 End Terminal]
//         Term 32 (EK1101) [EK1101 EtherCAT Coupler (2A E-Bus, ID switch)]
//           NDL1 (N1) (EL7047) [EL7047 1Ch. Stepper motor output stage (50V, 5A)]
//           NDL2 (N2) (EL7047) [EL7047 1Ch. Stepper motor output stage (50V, 5A)]
//           NDL3 (N3) (EL7047) [EL7047 1Ch. Stepper motor output stage (50V, 5A)]
//           NDL4 (N4) (EL7047) [EL7047 1Ch. Stepper motor output stage (50V, 5A)]
//           NTPA1 - NTPA2 (N6) (EL7342) [EL7342 2Ch. DC motor output stage (50V, 3.5A)]
//           NTPA3 - NTPA4 (N7) (EL7342) [EL7342 2Ch. DC motor output stage (50V, 3.5A)]
//           N8 (EL1008) [EL1008 8Ch. Dig. Input 24V, 3ms]
//           NTTA1 - NTTA2 (N9) (EL7342) [EL7342 2Ch. DC motor output stage (50V, 3.5A)]
//           NTTA3 - NTTA4 (N10) (EL7342) [EL7342 2Ch. DC motor output stage (50V, 3.5A)]
//           N11 (EL1008) [EL1008 8Ch. Dig. Input 24V, 3ms]
//           Power (N13) (EL9410) [EL9410 E-Bus Power Supplier  (Diagnostics)]
//           NTPB1 - NTPB2 (N14) (EL7342) [EL7342 2Ch. DC motor output stage (50V, 3.5A)]
//           NTPB3 - NTPB4 (N15) (EL7342) [EL7342 2Ch. DC motor output stage (50V, 3.5A)]
//           N16 (EL1008) [EL1008 8Ch. Dig. Input 24V, 3ms]
//           NTTB1 - NTTB2 (N18) (EL7342) [EL7342 2Ch. DC motor output stage (50V, 3.5A)]
//           NTTB3 - NTTB4 (N19) (EL7342) [EL7342 2Ch. DC motor output stage (50V, 3.5A)]
//           N20 (EL1008) [EL1008 8Ch. Dig. Input 24V, 3ms]
//           Term 53 (EL9011) [EL9011 End Terminal]
//       Term 50 (EM3701) [EM3701, 1Ch. differential pressure measuring terminal 100hPa (100mbar)]
//       Term 54 (EL9011) [EL9011 End Terminal]
// variable links:
//   NC-Task 1 SAF/Axes/NBS <-> Device 1 (EtherCAT)/Term 7 (EK1101)/Term 14 (EK1122)/Term 15 (EK1101)/NBS (N8) (EL7342)
//     Drive/Inputs/In/nState1 @bit 3 <-> DCM Status Channel 1/Status/Error
//     Drive/Inputs/In/nState1 @bit 5 <-> DCM Status Channel 1/Status/Moving negative
//     Drive/Inputs/In/nState1 @bit 4 <-> DCM Status Channel 1/Status/Moving positive
//     Drive/Inputs/In/nState1 @bit 1 <-> DCM Status Channel 1/Status/Ready
//     Drive/Inputs/In/nState1 <-> DCM Status Channel 1/Status/Ready to enable
//     Drive/Inputs/In/nState1 @bit 6 <-> DCM Status Channel 1/Status/Torque reduced
//     Drive/Inputs/In/nState1 @bit 2 <-> DCM Status Channel 1/Status/Warning
//     Drive/Inputs/In/nState2 @bit 3 <-> DCM Status Channel 1/Status/Digital input 1
//     Drive/Inputs/In/nState2 @bit 4 <-> DCM Status Channel 1/Status/Digital input 2
//     Drive/Inputs/In/nState2 @bit 5 <-> DCM Status Channel 1/Status/Sync error
//     Drive/Inputs/In/nState2 @bit 7 <-> DCM Status Channel 1/Status/TxPDO Toggle
//     Drive/Inputs/In/nState4 @bit 1 <-> WcState/InputToggle
//     Drive/Inputs/In/nState4 <-> WcState/WcState
//     Drive/Outputs/Out/nCtrl1 <-> DCM Control Channel 1/Control/Enable
//     Drive/Outputs/Out/nCtrl1 @bit 2 <-> DCM Control Channel 1/Control/Reduce torque
//     Drive/Outputs/Out/nCtrl1 @bit 1 <-> DCM Control Channel 1/Control/Reset
//     Drive/Outputs/Out/nCtrl1 @bit 3 <-> DCM Control Channel 1/Control/Threshold active
//     Drive/Outputs/Out/nDataOut2[0] <-> DCM Velocity Channel 1/Velocity
//     Enc/Inputs/In/nDataIn1[0] <-> ENC Status compact Channel 1/Counter value
//     Enc/Inputs/In/nDataIn2[0] <-> ENC Status compact Channel 1/Latch value
//     Enc/Inputs/In/nState1 @bit 4 <-> ENC Status compact Channel 1/Status/Counter overflow
//     Enc/Inputs/In/nState1 @bit 3 <-> ENC Status compact Channel 1/Status/Counter underflow
//     Enc/Inputs/In/nState1 @bit 7 <-> ENC Status compact Channel 1/Status/Extrapolation stall
//     Enc/Inputs/In/nState1 @bit 1 <-> ENC Status compact Channel 1/Status/Latch extern valid
//     Enc/Inputs/In/nState1 @bit 2 <-> ENC Status compact Channel 1/Status/Set counter done
//     Enc/Inputs/In/nState2 @bit 4 <-> ENC Status compact Channel 1/Status/Status of extern latch
//     Enc/Inputs/In/nState2 <-> ENC Status compact Channel 1/Status/Status of input A
//     Enc/Inputs/In/nState2 @bit 1 <-> ENC Status compact Channel 1/Status/Status of input B
//     Enc/Inputs/In/nState2 @bit 5 <-> ENC Status compact Channel 1/Status/Sync error
//     Enc/Inputs/In/nState2 @bit 7 <-> ENC Status compact Channel 1/Status/TxPDO Toggle
//     Enc/Inputs/In/nState4 @bit 1 <-> WcState/InputToggle
//     Enc/Inputs/In/nState4 <-> WcState/WcState
//     Enc/Outputs/Out/nCtrl1 @bit 3 <-> ENC Control compact Channel 1/Control/Enable latch extern on negative edge
//     Enc/Outputs/Out/nCtrl1 @bit 1 <-> ENC Control compact Channel 1/Control/Enable latch extern on positive edge
//     Enc/Outputs/Out/nCtrl1 @bit 2 <-> ENC Control compact Channel 1/Control/Set counter
//     Enc/Outputs/Out/nDataOut1[0] <-> ENC Control compact Channel 1/Set counter value
//   NC-Task 1 SAF/Axes/NCP1 <-> Device 1 (EtherCAT)/Term 7 (EK1101)/Term 14 (EK1122)/Term 15 (EK1101)/NCP1 - NCP2 (N1) (EL7342)
//     Drive/Inputs/In/nState1 @bit 3 <-> DCM Status Channel 1/Status/Error
//     Drive/Inputs/In/nState1 @bit 5 <-> DCM Status Channel 1/Status/Moving negative
//     Drive/Inputs/In/nState1 @bit 4 <-> DCM Status Channel 1/Status/Moving positive
//     Drive/Inputs/In/nState1 @bit 1 <-> DCM Status Channel 1/Status/Ready
//     Drive/Inputs/In/nState1 <-> DCM Status Channel 1/Status/Ready to enable
//     Drive/Inputs/In/nState1 @bit 6 <-> DCM Status Channel 1/Status/Torque reduced
//     Drive/Inputs/In/nState1 @bit 2 <-> DCM Status Channel 1/Status/Warning
//     Drive/Inputs/In/nState2 @bit 3 <-> DCM Status Channel 1/Status/Digital input 1
//     Drive/Inputs/In/nState2 @bit 4 <-> DCM Status Channel 1/Status/Digital input 2
//     Drive/Inputs/In/nState2 @bit 5 <-> DCM Status Channel 1/Status/Sync error
//     Drive/Inputs/In/nState2 @bit 7 <-> DCM Status Channel 1/Status/TxPDO Toggle
//     Drive/Inputs/In/nState4 @bit 1 <-> WcState/InputToggle
//     Drive/Inputs/In/nState4 <-> WcState/WcState
//     Drive/Outputs/Out/nCtrl1 <-> DCM Control Channel 1/Control/Enable
//     Drive/Outputs/Out/nCtrl1 @bit 2 <-> DCM Control Channel 1/Control/Reduce torque
//     Drive/Outputs/Out/nCtrl1 @bit 1 <-> DCM Control Channel 1/Control/Reset
//     Drive/Outputs/Out/nCtrl1 @bit 3 <-> DCM Control Channel 1/Control/Threshold active
//     Drive/Outputs/Out/nDataOut2[0] <-> DCM Velocity Channel 1/Velocity
//     Enc/Inputs/In/nDataIn1[0] <-> ENC Status compact Channel 1/Counter value
//     Enc/Inputs/In/nDataIn2[0] <-> ENC Status compact Channel 1/Latch value
//     Enc/Inputs/In/nState1 @bit 4 <-> ENC Status compact Channel 1/Status/Counter overflow
//     Enc/Inputs/In/nState1 @bit 3 <-> ENC Status compact Channel 1/Status/Counter underflow
//     Enc/Inputs/In/nState1 @bit 7 <-> ENC Status compact Channel 1/Status/Extrapolation stall
//     Enc/Inputs/In/nState1 @bit 1 <-> ENC Status compact Channel 1/Status/Latch extern valid
//     Enc/Inputs/In/nState1 @bit 2 <-> ENC Status compact Channel 1/Status/Set counter done
//     Enc/Inputs/In/nState2 @bit 4 <-> ENC Status compact Channel 1/Status/Status of extern latch
//     Enc/Inputs/In/nState2 <-> ENC Status compact Channel 1/Status/Status of input A
//     Enc/Inputs/In/nState2 @bit 1 <-> ENC Status compact Channel 1/Status/Status of input B
//     Enc/Inputs/In/nState2 @bit 5 <-> ENC Status compact Channel 1/Status/Sync error
//     Enc/Inputs/In/nState2 @bit 7 <-> ENC Status compact Channel 1/Status/TxPDO Toggle
//     Enc/Inputs/In/nState4 @bit 1 <-> WcState/InputToggle
//     Enc/Inputs/In/nState4 <-> WcState/WcState
//     Enc/Outputs/Out/nCtrl1 @bit 3 <-> ENC Control compact Channel 1/Control/Enable latch extern on negative edge
//     Enc/Outputs/Out/nCtrl1 @bit 1 <-> ENC Control compact Channel 1/Control/Enable latch extern on positive edge
//     Enc/Outputs/Out/nCtrl1 @bit 2 <-> ENC Control compact Channel 1/Control/Set counter
//     Enc/Outputs/Out/nDataOut1[0] <-> ENC Control compact Channel 1/Set counter value
//   NC-Task 1 SAF/Axes/NCP2 <-> Device 1 (EtherCAT)/Term 7 (EK1101)/Term 14 (EK1122)/Term 15 (EK1101)/NCP1 - NCP2 (N1) (EL7342)
//     Drive/Inputs/In/nState1 @bit 3 <-> DCM Status Channel 2/Status/Error
//     Drive/Inputs/In/nState1 @bit 5 <-> DCM Status Channel 2/Status/Moving negative
//     Drive/Inputs/In/nState1 @bit 4 <-> DCM Status Channel 2/Status/Moving positive
//     Drive/Inputs/In/nState1 @bit 1 <-> DCM Status Channel 2/Status/Ready
//     Drive/Inputs/In/nState1 <-> DCM Status Channel 2/Status/Ready to enable
//     Drive/Inputs/In/nState1 @bit 6 <-> DCM Status Channel 2/Status/Torque reduced
//     Drive/Inputs/In/nState1 @bit 2 <-> DCM Status Channel 2/Status/Warning
//     Drive/Inputs/In/nState2 @bit 3 <-> DCM Status Channel 2/Status/Digital input 1
//     Drive/Inputs/In/nState2 @bit 4 <-> DCM Status Channel 2/Status/Digital input 2
//     Drive/Inputs/In/nState2 @bit 5 <-> DCM Status Channel 2/Status/Sync error
//     Drive/Inputs/In/nState2 @bit 7 <-> DCM Status Channel 2/Status/TxPDO Toggle
//     Drive/Inputs/In/nState4 @bit 1 <-> WcState/InputToggle
//     Drive/Inputs/In/nState4 <-> WcState/WcState
//     Drive/Outputs/Out/nCtrl1 <-> DCM Control Channel 2/Control/Enable
//     Drive/Outputs/Out/nCtrl1 @bit 2 <-> DCM Control Channel 2/Control/Reduce torque
//     Drive/Outputs/Out/nCtrl1 @bit 1 <-> DCM Control Channel 2/Control/Reset
//     Drive/Outputs/Out/nCtrl1 @bit 3 <-> DCM Control Channel 2/Control/Threshold active
//     Drive/Outputs/Out/nDataOut2[0] <-> DCM Velocity Channel 2/Velocity
//     Enc/Inputs/In/nDataIn1[0] <-> ENC Status compact Channel 2/Counter value
//     Enc/Inputs/In/nDataIn2[0] <-> ENC Status compact Channel 2/Latch value
//     Enc/Inputs/In/nState1 @bit 4 <-> ENC Status compact Channel 2/Status/Counter overflow
//     Enc/Inputs/In/nState1 @bit 3 <-> ENC Status compact Channel 2/Status/Counter underflow
//     Enc/Inputs/In/nState1 @bit 7 <-> ENC Status compact Channel 2/Status/Extrapolation stall
//     Enc/Inputs/In/nState1 @bit 1 <-> ENC Status compact Channel 2/Status/Latch extern valid
//     Enc/Inputs/In/nState1 @bit 2 <-> ENC Status compact Channel 2/Status/Set counter done
//     Enc/Inputs/In/nState2 @bit 4 <-> ENC Status compact Channel 2/Status/Status of extern latch
//     Enc/Inputs/In/nState2 <-> ENC Status compact Channel 2/Status/Status of input A
//     Enc/Inputs/In/nState2 @bit 1 <-> ENC Status compact Channel 2/Status/Status of input B
//     Enc/Inputs/In/nState2 @bit 5 <-> ENC Status compact Channel 2/Status/Sync error
//     Enc/Inputs/In/nState2 @bit 7 <-> ENC Status compact Channel 2/Status/TxPDO Toggle
//     Enc/Inputs/In/nState4 @bit 1 <-> WcState/InputToggle
//     Enc/Inputs/In/nState4 <-> WcState/WcState
//     Enc/Outputs/Out/nCtrl1 @bit 3 <-> ENC Control compact Channel 2/Control/Enable latch extern on negative edge
//     Enc/Outputs/Out/nCtrl1 @bit 1 <-> ENC Control compact Channel 2/Control/Enable latch extern on positive edge
//     Enc/Outputs/Out/nCtrl1 @bit 2 <-> ENC Control compact Channel 2/Control/Set counter
//     Enc/Outputs/Out/nDataOut1[0] <-> ENC Control compact Channel 2/Set counter value
//   NC-Task 1 SAF/Axes/NCP3 <-> Device 1 (EtherCAT)/Term 7 (EK1101)/Term 14 (EK1122)/Term 15 (EK1101)/NCP3 - NCP4 (N2) (EL7342)
//     Drive/Inputs/In/nState1 @bit 3 <-> DCM Status Channel 1/Status/Error
//     Drive/Inputs/In/nState1 @bit 5 <-> DCM Status Channel 1/Status/Moving negative
//     Drive/Inputs/In/nState1 @bit 4 <-> DCM Status Channel 1/Status/Moving positive
//     Drive/Inputs/In/nState1 @bit 1 <-> DCM Status Channel 1/Status/Ready
//     Drive/Inputs/In/nState1 <-> DCM Status Channel 1/Status/Ready to enable
//     Drive/Inputs/In/nState1 @bit 6 <-> DCM Status Channel 1/Status/Torque reduced
//     Drive/Inputs/In/nState1 @bit 2 <-> DCM Status Channel 1/Status/Warning
//     Drive/Inputs/In/nState2 @bit 3 <-> DCM Status Channel 1/Status/Digital input 1
//     Drive/Inputs/In/nState2 @bit 4 <-> DCM Status Channel 1/Status/Digital input 2
//     Drive/Inputs/In/nState2 @bit 5 <-> DCM Status Channel 1/Status/Sync error
//     Drive/Inputs/In/nState2 @bit 7 <-> DCM Status Channel 1/Status/TxPDO Toggle
//     Drive/Inputs/In/nState4 @bit 1 <-> WcState/InputToggle
//     Drive/Inputs/In/nState4 <-> WcState/WcState
//     Drive/Outputs/Out/nCtrl1 <-> DCM Control Channel 1/Control/Enable
//     Drive/Outputs/Out/nCtrl1 @bit 2 <-> DCM Control Channel 1/Control/Reduce torque
//     Drive/Outputs/Out/nCtrl1 @bit 1 <-> DCM Control Channel 1/Control/Reset
//     Drive/Outputs/Out/nCtrl1 @bit 3 <-> DCM Control Channel 1/Control/Threshold active
//     Drive/Outputs/Out/nDataOut2[0] <-> DCM Velocity Channel 1/Velocity
//     Enc/Inputs/In/nDataIn1[0] <-> ENC Status compact Channel 1/Counter value
//     Enc/Inputs/In/nDataIn2[0] <-> ENC Status compact Channel 1/Latch value
//     Enc/Inputs/In/nState1 @bit 4 <-> ENC Status compact Channel 1/Status/Counter overflow
//     Enc/Inputs/In/nState1 @bit 3 <-> ENC Status compact Channel 1/Status/Counter underflow
//     Enc/Inputs/In/nState1 @bit 7 <-> ENC Status compact Channel 1/Status/Extrapolation stall
//     Enc/Inputs/In/nState1 @bit 1 <-> ENC Status compact Channel 1/Status/Latch extern valid
//     Enc/Inputs/In/nState1 @bit 2 <-> ENC Status compact Channel 1/Status/Set counter done
//     Enc/Inputs/In/nState2 @bit 4 <-> ENC Status compact Channel 1/Status/Status of extern latch
//     Enc/Inputs/In/nState2 <-> ENC Status compact Channel 1/Status/Status of input A
//     Enc/Inputs/In/nState2 @bit 1 <-> ENC Status compact Channel 1/Status/Status of input B
//     Enc/Inputs/In/nState2 @bit 5 <-> ENC Status compact Channel 1/Status/Sync error
//     Enc/Inputs/In/nState2 @bit 7 <-> ENC Status compact Channel 1/Status/TxPDO Toggle
//     Enc/Inputs/In/nState4 @bit 1 <-> WcState/InputToggle
//     Enc/Inputs/In/nState4 <-> WcState/WcState
//     Enc/Outputs/Out/nCtrl1 @bit 3 <-> ENC Control compact Channel 1/Control/Enable latch extern on negative edge
//     Enc/Outputs/Out/nCtrl1 @bit 1 <-> ENC Control compact Channel 1/Control/Enable latch extern on positive edge
//     Enc/Outputs/Out/nCtrl1 @bit 2 <-> ENC Control compact Channel 1/Control/Set counter
//     Enc/Outputs/Out/nDataOut1[0] <-> ENC Control compact Channel 1/Set counter value
//   NC-Task 1 SAF/Axes/NCP4 <-> Device 1 (EtherCAT)/Term 7 (EK1101)/Term 14 (EK1122)/Term 15 (EK1101)/NCP3 - NCP4 (N2) (EL7342)
//     Drive/Inputs/In/nState1 @bit 3 <-> DCM Status Channel 2/Status/Error
//     Drive/Inputs/In/nState1 @bit 5 <-> DCM Status Channel 2/Status/Moving negative
//     Drive/Inputs/In/nState1 @bit 4 <-> DCM Status Channel 2/Status/Moving positive
//     Drive/Inputs/In/nState1 @bit 1 <-> DCM Status Channel 2/Status/Ready
//     Drive/Inputs/In/nState1 <-> DCM Status Channel 2/Status/Ready to enable
//     Drive/Inputs/In/nState1 @bit 6 <-> DCM Status Channel 2/Status/Torque reduced
//     Drive/Inputs/In/nState1 @bit 2 <-> DCM Status Channel 2/Status/Warning
//     Drive/Inputs/In/nState2 @bit 3 <-> DCM Status Channel 2/Status/Digital input 1
//     Drive/Inputs/In/nState2 @bit 4 <-> DCM Status Channel 2/Status/Digital input 2
//     Drive/Inputs/In/nState2 @bit 5 <-> DCM Status Channel 2/Status/Sync error
//     Drive/Inputs/In/nState2 @bit 7 <-> DCM Status Channel 2/Status/TxPDO Toggle
//     Drive/Inputs/In/nState4 @bit 1 <-> WcState/InputToggle
//     Drive/Inputs/In/nState4 <-> WcState/WcState
//     Drive/Outputs/Out/nCtrl1 <-> DCM Control Channel 2/Control/Enable
//     Drive/Outputs/Out/nCtrl1 @bit 2 <-> DCM Control Channel 2/Control/Reduce torque
//     Drive/Outputs/Out/nCtrl1 @bit 1 <-> DCM Control Channel 2/Control/Reset
//     Drive/Outputs/Out/nCtrl1 @bit 3 <-> DCM Control Channel 2/Control/Threshold active
//     Drive/Outputs/Out/nDataOut2[0] <-> DCM Velocity Channel 2/Velocity
//     Enc/Inputs/In/nDataIn1[0] <-> ENC Status compact Channel 2/Counter value
//     Enc/Inputs/In/nDataIn2[0] <-> ENC Status compact Channel 2/Latch value
//     Enc/Inputs/In/nState1 @bit 4 <-> ENC Status compact Channel 2/Status/Counter overflow
//     Enc/Inputs/In/nState1 @bit 3 <-> ENC Status compact Channel 2/Status/Counter underflow
//     Enc/Inputs/In/nState1 @bit 7 <-> ENC Status compact Channel 2/Status/Extrapolation stall
//     Enc/Inputs/In/nState1 @bit 1 <-> ENC Status compact Channel 2/Status/Latch extern valid
//     Enc/Inputs/In/nState1 @bit 2 <-> ENC Status compact Channel 2/Status/Set counter done
//     Enc/Inputs/In/nState2 @bit 4 <-> ENC Status compact Channel 2/Status/Status of extern latch
//     Enc/Inputs/In/nState2 <-> ENC Status compact Channel 2/Status/Status of input A
//     Enc/Inputs/In/nState2 @bit 1 <-> ENC Status compact Channel 2/Status/Status of input B
//     Enc/Inputs/In/nState2 @bit 5 <-> ENC Status compact Channel 2/Status/Sync error
//     Enc/Inputs/In/nState2 @bit 7 <-> ENC Status compact Channel 2/Status/TxPDO Toggle
//     Enc/Inputs/In/nState4 @bit 1 <-> WcState/InputToggle
//     Enc/Inputs/In/nState4 <-> WcState/WcState
//     Enc/Outputs/Out/nCtrl1 @bit 3 <-> ENC Control compact Channel 2/Control/Enable latch extern on negative edge
//     Enc/Outputs/Out/nCtrl1 @bit 1 <-> ENC Control compact Channel 2/Control/Enable latch extern on positive edge
//     Enc/Outputs/Out/nCtrl1 @bit 2 <-> ENC Control compact Channel 2/Control/Set counter
//     Enc/Outputs/Out/nDataOut1[0] <-> ENC Control compact Channel 2/Set counter value
//   NC-Task 1 SAF/Axes/NDL1 <-> Device 1 (EtherCAT)/Term 7 (EK1101)/Term 14 (EK1122)/Term 32 (EK1101)/NDL1 (N1) (EL7047)
//     Drive/Inputs/In/nState1 @bit 3 <-> STM Status/Status/Error
//     Drive/Inputs/In/nState1 @bit 7 <-> STM Status/Status/Motor stall
//     Drive/Inputs/In/nState1 @bit 5 <-> STM Status/Status/Moving negative
//     Drive/Inputs/In/nState1 @bit 4 <-> STM Status/Status/Moving positive
//     Drive/Inputs/In/nState1 @bit 1 <-> STM Status/Status/Ready
//     Drive/Inputs/In/nState1 <-> STM Status/Status/Ready to enable
//     Drive/Inputs/In/nState1 @bit 6 <-> STM Status/Status/Torque reduced
//     Drive/Inputs/In/nState1 @bit 2 <-> STM Status/Status/Warning
//     Drive/Inputs/In/nState2 @bit 3 <-> STM Status/Status/Digital input 1
//     Drive/Inputs/In/nState2 @bit 4 <-> STM Status/Status/Digital input 2
//     Drive/Inputs/In/nState2 @bit 5 <-> STM Status/Status/Sync error
//     Drive/Inputs/In/nState2 @bit 7 <-> STM Status/Status/TxPDO Toggle
//     Drive/Inputs/In/nState4 @bit 1 <-> WcState/InputToggle
//     Drive/Inputs/In/nState4 <-> WcState/WcState
//     Drive/Outputs/Out/nCtrl1 <-> STM Control/Control/Enable
//     Drive/Outputs/Out/nCtrl1 @bit 2 <-> STM Control/Control/Reduce torque
//     Drive/Outputs/Out/nCtrl1 @bit 1 <-> STM Control/Control/Reset
//     Drive/Outputs/Out/nCtrl2 @bit 3 <-> STM Control/Control/Digital output 1
//     Drive/Outputs/Out/nDataOut2[0] <-> STM Velocity/Velocity
//     Enc/Inputs/In/nDataIn1[0] <-> ENC Status compact/Counter value
//     Enc/Inputs/In/nDataIn2[0] <-> ENC Status compact/Latch value
//     Enc/Inputs/In/nState1 @bit 4 <-> ENC Status compact/Status/Counter overflow
//     Enc/Inputs/In/nState1 @bit 3 <-> ENC Status compact/Status/Counter underflow
//     Enc/Inputs/In/nState1 @bit 7 <-> ENC Status compact/Status/Extrapolation stall
//     Enc/Inputs/In/nState1 <-> ENC Status compact/Status/Latch C valid
//     Enc/Inputs/In/nState1 @bit 1 <-> ENC Status compact/Status/Latch extern valid
//     Enc/Inputs/In/nState1 @bit 2 <-> ENC Status compact/Status/Set counter done
//     Enc/Inputs/In/nState2 @bit 4 <-> ENC Status compact/Status/Status of extern latch
//     Enc/Inputs/In/nState2 <-> ENC Status compact/Status/Status of input A
//     Enc/Inputs/In/nState2 @bit 1 <-> ENC Status compact/Status/Status of input B
//     Enc/Inputs/In/nState2 @bit 2 <-> ENC Status compact/Status/Status of input C
//     Enc/Inputs/In/nState2 @bit 5 <-> ENC Status compact/Status/Sync error
//     Enc/Inputs/In/nState2 @bit 7 <-> ENC Status compact/Status/TxPDO Toggle
//     Enc/Inputs/In/nState4 @bit 1 <-> WcState/InputToggle
//     Enc/Inputs/In/nState4 <-> WcState/WcState
//     Enc/Outputs/Out/nCtrl1 <-> ENC Control compact/Control/Enable latch C
//     Enc/Outputs/Out/nCtrl1 @bit 3 <-> ENC Control compact/Control/Enable latch extern on negative edge
//     Enc/Outputs/Out/nCtrl1 @bit 1 <-> ENC Control compact/Control/Enable latch extern on positive edge
//     Enc/Outputs/Out/nCtrl1 @bit 2 <-> ENC Control compact/Control/Set counter
//     Enc/Outputs/Out/nDataOut1[0] <-> ENC Control compact/Set counter value
//   NC-Task 1 SAF/Axes/NDL2 <-> Device 1 (EtherCAT)/Term 7 (EK1101)/Term 14 (EK1122)/Term 32 (EK1101)/NDL2 (N2) (EL7047)
//     Drive/Inputs/In/nState1 @bit 3 <-> STM Status/Status/Error
//     Drive/Inputs/In/nState1 @bit 7 <-> STM Status/Status/Motor stall
//     Drive/Inputs/In/nState1 @bit 5 <-> STM Status/Status/Moving negative
//     Drive/Inputs/In/nState1 @bit 4 <-> STM Status/Status/Moving positive
//     Drive/Inputs/In/nState1 @bit 1 <-> STM Status/Status/Ready
//     Drive/Inputs/In/nState1 <-> STM Status/Status/Ready to enable
//     Drive/Inputs/In/nState1 @bit 6 <-> STM Status/Status/Torque reduced
//     Drive/Inputs/In/nState1 @bit 2 <-> STM Status/Status/Warning
//     Drive/Inputs/In/nState2 @bit 3 <-> STM Status/Status/Digital input 1
//     Drive/Inputs/In/nState2 @bit 4 <-> STM Status/Status/Digital input 2
//     Drive/Inputs/In/nState2 @bit 5 <-> STM Status/Status/Sync error
//     Drive/Inputs/In/nState2 @bit 7 <-> STM Status/Status/TxPDO Toggle
//     Drive/Inputs/In/nState4 @bit 1 <-> WcState/InputToggle
//     Drive/Inputs/In/nState4 <-> WcState/WcState
//     Drive/Outputs/Out/nCtrl1 <-> STM Control/Control/Enable
//     Drive/Outputs/Out/nCtrl1 @bit 2 <-> STM Control/Control/Reduce torque
//     Drive/Outputs/Out/nCtrl1 @bit 1 <-> STM Control/Control/Reset
//     Drive/Outputs/Out/nCtrl2 @bit 3 <-> STM Control/Control/Digital output 1
//     Drive/Outputs/Out/nDataOut2[0] <-> STM Velocity/Velocity
//     Enc/Inputs/In/nDataIn1[0] <-> ENC Status compact/Counter value
//     Enc/Inputs/In/nDataIn2[0] <-> ENC Status compact/Latch value
//     Enc/Inputs/In/nState1 @bit 4 <-> ENC Status compact/Status/Counter overflow
//     Enc/Inputs/In/nState1 @bit 3 <-> ENC Status compact/Status/Counter underflow
//     Enc/Inputs/In/nState1 @bit 7 <-> ENC Status compact/Status/Extrapolation stall
//     Enc/Inputs/In/nState1 <-> ENC Status compact/Status/Latch C valid
//     Enc/Inputs/In/nState1 @bit 1 <-> ENC Status compact/Status/Latch extern valid
//     Enc/Inputs/In/nState1 @bit 2 <-> ENC Status compact/Status/Set counter done
//     Enc/Inputs/In/nState2 @bit 4 <-> ENC Status compact/Status/Status of extern latch
//     Enc/Inputs/In/nState2 <-> ENC Status compact/Status/Status of input A
//     Enc/Inputs/In/nState2 @bit 1 <-> ENC Status compact/Status/Status of input B
//     Enc/Inputs/In/nState2 @bit 2 <-> ENC Status compact/Status/Status of input C
//     Enc/Inputs/In/nState2 @bit 5 <-> ENC Status compact/Status/Sync error
//     Enc/Inputs/In/nState2 @bit 7 <-> ENC Status compact/Status/TxPDO Toggle
//     Enc/Inputs/In/nState4 @bit 1 <-> WcState/InputToggle
//     Enc/Inputs/In/nState4 <-> WcState/WcState
//     Enc/Outputs/Out/nCtrl1 <-> ENC Control compact/Control/Enable latch C
//     Enc/Outputs/Out/nCtrl1 @bit 3 <-> ENC Control compact/Control/Enable latch extern on negative edge
//     Enc/Outputs/Out/nCtrl1 @bit 1 <-> ENC Control compact/Control/Enable latch extern on positive edge
//     Enc/Outputs/Out/nCtrl1 @bit 2 <-> ENC Control compact/Control/Set counter
//     Enc/Outputs/Out/nDataOut1[0] <-> ENC Control compact/Set counter value
//   NC-Task 1 SAF/Axes/NDL3 <-> Device 1 (EtherCAT)/Term 7 (EK1101)/Term 14 (EK1122)/Term 32 (EK1101)/NDL3 (N3) (EL7047)
//     Drive/Inputs/In/nState1 @bit 3 <-> STM Status/Status/Error
//     Drive/Inputs/In/nState1 @bit 7 <-> STM Status/Status/Motor stall
//     Drive/Inputs/In/nState1 @bit 5 <-> STM Status/Status/Moving negative
//     Drive/Inputs/In/nState1 @bit 4 <-> STM Status/Status/Moving positive
//     Drive/Inputs/In/nState1 @bit 1 <-> STM Status/Status/Ready
//     Drive/Inputs/In/nState1 <-> STM Status/Status/Ready to enable
//     Drive/Inputs/In/nState1 @bit 6 <-> STM Status/Status/Torque reduced
//     Drive/Inputs/In/nState1 @bit 2 <-> STM Status/Status/Warning
//     Drive/Inputs/In/nState2 @bit 3 <-> STM Status/Status/Digital input 1
//     Drive/Inputs/In/nState2 @bit 4 <-> STM Status/Status/Digital input 2
//     Drive/Inputs/In/nState2 @bit 5 <-> STM Status/Status/Sync error
//     Drive/Inputs/In/nState2 @bit 7 <-> STM Status/Status/TxPDO Toggle
//     Drive/Inputs/In/nState4 @bit 1 <-> WcState/InputToggle
//     Drive/Inputs/In/nState4 <-> WcState/WcState
//     Drive/Outputs/Out/nCtrl1 <-> STM Control/Control/Enable
//     Drive/Outputs/Out/nCtrl1 @bit 2 <-> STM Control/Control/Reduce torque
//     Drive/Outputs/Out/nCtrl1 @bit 1 <-> STM Control/Control/Reset
//     Drive/Outputs/Out/nCtrl2 @bit 3 <-> STM Control/Control/Digital output 1
//     Drive/Outputs/Out/nDataOut2[0] <-> STM Velocity/Velocity
//     Enc/Inputs/In/nDataIn1[0] <-> ENC Status compact/Counter value
//     Enc/Inputs/In/nDataIn2[0] <-> ENC Status compact/Latch value
//     Enc/Inputs/In/nState1 @bit 4 <-> ENC Status compact/Status/Counter overflow
//     Enc/Inputs/In/nState1 @bit 3 <-> ENC Status compact/Status/Counter underflow
//     Enc/Inputs/In/nState1 @bit 7 <-> ENC Status compact/Status/Extrapolation stall
//     Enc/Inputs/In/nState1 <-> ENC Status compact/Status/Latch C valid
//     Enc/Inputs/In/nState1 @bit 1 <-> ENC Status compact/Status/Latch extern valid
//     Enc/Inputs/In/nState1 @bit 2 <-> ENC Status compact/Status/Set counter done
//     Enc/Inputs/In/nState2 @bit 4 <-> ENC Status compact/Status/Status of extern latch
//     Enc/Inputs/In/nState2 <-> ENC Status compact/Status/Status of input A
//     Enc/Inputs/In/nState2 @bit 1 <-> ENC Status compact/Status/Status of input B
//     Enc/Inputs/In/nState2 @bit 2 <-> ENC Status compact/Status/Status of input C
//     Enc/Inputs/In/nState2 @bit 5 <-> ENC Status compact/Status/Sync error
//     Enc/Inputs/In/nState2 @bit 7 <-> ENC Status compact/Status/TxPDO Toggle
//     Enc/Inputs/In/nState4 @bit 1 <-> WcState/InputToggle
//     Enc/Inputs/In/nState4 <-> WcState/WcState
//     Enc/Outputs/Out/nCtrl1 <-> ENC Control compact/Control/Enable latch C
//     Enc/Outputs/Out/nCtrl1 @bit 3 <-> ENC Control compact/Control/Enable latch extern on negative edge
//     Enc/Outputs/Out/nCtrl1 @bit 1 <-> ENC Control compact/Control/Enable latch extern on positive edge
//     Enc/Outputs/Out/nCtrl1 @bit 2 <-> ENC Control compact/Control/Set counter
//     Enc/Outputs/Out/nDataOut1[0] <-> ENC Control compact/Set counter value
//   NC-Task 1 SAF/Axes/NDL4 <-> Device 1 (EtherCAT)/Term 7 (EK1101)/Term 14 (EK1122)/Term 32 (EK1101)/NDL4 (N4) (EL7047)
//     Drive/Inputs/In/nState1 @bit 3 <-> STM Status/Status/Error
//     Drive/Inputs/In/nState1 @bit 7 <-> STM Status/Status/Motor stall
//     Drive/Inputs/In/nState1 @bit 5 <-> STM Status/Status/Moving negative
//     Drive/Inputs/In/nState1 @bit 4 <-> STM Status/Status/Moving positive
//     Drive/Inputs/In/nState1 @bit 1 <-> STM Status/Status/Ready
//     Drive/Inputs/In/nState1 <-> STM Status/Status/Ready to enable
//     Drive/Inputs/In/nState1 @bit 6 <-> STM Status/Status/Torque reduced
//     Drive/Inputs/In/nState1 @bit 2 <-> STM Status/Status/Warning
//     Drive/Inputs/In/nState2 @bit 3 <-> STM Status/Status/Digital input 1
//     Drive/Inputs/In/nState2 @bit 4 <-> STM Status/Status/Digital input 2
//     Drive/Inputs/In/nState2 @bit 5 <-> STM Status/Status/Sync error
//     Drive/Inputs/In/nState2 @bit 7 <-> STM Status/Status/TxPDO Toggle
//     Drive/Inputs/In/nState4 @bit 1 <-> WcState/InputToggle
//     Drive/Inputs/In/nState4 <-> WcState/WcState
//     Drive/Outputs/Out/nCtrl1 <-> STM Control/Control/Enable
//     Drive/Outputs/Out/nCtrl1 @bit 2 <-> STM Control/Control/Reduce torque
//     Drive/Outputs/Out/nCtrl1 @bit 1 <-> STM Control/Control/Reset
//     Drive/Outputs/Out/nCtrl2 @bit 3 <-> STM Control/Control/Digital output 1
//     Drive/Outputs/Out/nDataOut2[0] <-> STM Velocity/Velocity
//     Enc/Inputs/In/nDataIn1[0] <-> ENC Status compact/Counter value
//     Enc/Inputs/In/nDataIn2[0] <-> ENC Status compact/Latch value
//     Enc/Inputs/In/nState1 @bit 4 <-> ENC Status compact/Status/Counter overflow
//     Enc/Inputs/In/nState1 @bit 3 <-> ENC Status compact/Status/Counter underflow
//     Enc/Inputs/In/nState1 @bit 7 <-> ENC Status compact/Status/Extrapolation stall
//     Enc/Inputs/In/nState1 <-> ENC Status compact/Status/Latch C valid
//     Enc/Inputs/In/nState1 @bit 1 <-> ENC Status compact/Status/Latch extern valid
//     Enc/Inputs/In/nState1 @bit 2 <-> ENC Status compact/Status/Set counter done
//     Enc/Inputs/In/nState2 @bit 4 <-> ENC Status compact/Status/Status of extern latch
//     Enc/Inputs/In/nState2 <-> ENC Status compact/Status/Status of input A
//     Enc/Inputs/In/nState2 @bit 1 <-> ENC Status compact/Status/Status of input B
//     Enc/Inputs/In/nState2 @bit 2 <-> ENC Status compact/Status/Status of input C
//     Enc/Inputs/In/nState2 @bit 5 <-> ENC Status compact/Status/Sync error
//     Enc/Inputs/In/nState2 @bit 7 <-> ENC Status compact/Status/TxPDO Toggle
//     Enc/Inputs/In/nState4 @bit 1 <-> WcState/InputToggle
//     Enc/Inputs/In/nState4 <-> WcState/WcState
//     Enc/Outputs/Out/nCtrl1 <-> ENC Control compact/Control/Enable latch C
//     Enc/Outputs/Out/nCtrl1 @bit 3 <-> ENC Control compact/Control/Enable latch extern on negative edge
//     Enc/Outputs/Out/nCtrl1 @bit 1 <-> ENC Control compact/Control/Enable latch extern on positive edge
//     Enc/Outputs/Out/nCtrl1 @bit 2 <-> ENC Control compact/Control/Set counter
//     Enc/Outputs/Out/nDataOut1[0] <-> ENC Control compact/Set counter value
//   NC-Task 1 SAF/Axes/NGP1 <-> Device 1 (EtherCAT)/Term 7 (EK1101)/Term 14 (EK1122)/Term 15 (EK1101)/NGP1 - NGP2 (N5) (EL7342)
//     Drive/Inputs/In/nState1 @bit 3 <-> DCM Status Channel 1/Status/Error
//     Drive/Inputs/In/nState1 @bit 5 <-> DCM Status Channel 1/Status/Moving negative
//     Drive/Inputs/In/nState1 @bit 4 <-> DCM Status Channel 1/Status/Moving positive
//     Drive/Inputs/In/nState1 @bit 1 <-> DCM Status Channel 1/Status/Ready
//     Drive/Inputs/In/nState1 <-> DCM Status Channel 1/Status/Ready to enable
//     Drive/Inputs/In/nState1 @bit 6 <-> DCM Status Channel 1/Status/Torque reduced
//     Drive/Inputs/In/nState1 @bit 2 <-> DCM Status Channel 1/Status/Warning
//     Drive/Inputs/In/nState2 @bit 3 <-> DCM Status Channel 1/Status/Digital input 1
//     Drive/Inputs/In/nState2 @bit 4 <-> DCM Status Channel 1/Status/Digital input 2
//     Drive/Inputs/In/nState4 @bit 1 <-> WcState/InputToggle
//     Drive/Inputs/In/nState4 <-> WcState/WcState
//     Drive/Outputs/Out/nCtrl1 <-> DCM Control Channel 1/Control/Enable
//     Drive/Outputs/Out/nCtrl1 @bit 2 <-> DCM Control Channel 1/Control/Reduce torque
//     Drive/Outputs/Out/nCtrl1 @bit 1 <-> DCM Control Channel 1/Control/Reset
//     Drive/Outputs/Out/nDataOut2[0] <-> DCM Velocity Channel 1/Velocity
//     Enc/Inputs/In/nDataIn1[0] <-> ENC Status compact Channel 1/Counter value
//     Enc/Inputs/In/nDataIn2[0] <-> ENC Status compact Channel 1/Latch value
//     Enc/Inputs/In/nState1 @bit 4 <-> ENC Status compact Channel 1/Status/Counter overflow
//     Enc/Inputs/In/nState1 @bit 3 <-> ENC Status compact Channel 1/Status/Counter underflow
//     Enc/Inputs/In/nState1 @bit 7 <-> ENC Status compact Channel 1/Status/Extrapolation stall
//     Enc/Inputs/In/nState1 @bit 1 <-> ENC Status compact Channel 1/Status/Latch extern valid
//     Enc/Inputs/In/nState1 @bit 2 <-> ENC Status compact Channel 1/Status/Set counter done
//     Enc/Inputs/In/nState2 @bit 4 <-> ENC Status compact Channel 1/Status/Status of extern latch
//     Enc/Inputs/In/nState2 <-> ENC Status compact Channel 1/Status/Status of input A
//     Enc/Inputs/In/nState2 @bit 1 <-> ENC Status compact Channel 1/Status/Status of input B
//     Enc/Inputs/In/nState4 @bit 1 <-> WcState/InputToggle
//     Enc/Inputs/In/nState4 <-> WcState/WcState
//     Enc/Outputs/Out/nCtrl1 @bit 3 <-> ENC Control compact Channel 1/Control/Enable latch extern on negative edge
//     Enc/Outputs/Out/nCtrl1 @bit 1 <-> ENC Control compact Channel 1/Control/Enable latch extern on positive edge
//     Enc/Outputs/Out/nCtrl1 @bit 2 <-> ENC Control compact Channel 1/Control/Set counter
//     Enc/Outputs/Out/nDataOut1[0] <-> ENC Control compact Channel 1/Set counter value
//   NC-Task 1 SAF/Axes/NGP2 <-> Device 1 (EtherCAT)/Term 7 (EK1101)/Term 14 (EK1122)/Term 15 (EK1101)/NGP1 - NGP2 (N5) (EL7342)
//     Drive/Inputs/In/nState1 @bit 3 <-> DCM Status Channel 2/Status/Error
//     Drive/Inputs/In/nState1 @bit 5 <-> DCM Status Channel 2/Status/Moving negative
//     Drive/Inputs/In/nState1 @bit 4 <-> DCM Status Channel 2/Status/Moving positive
//     Drive/Inputs/In/nState1 @bit 1 <-> DCM Status Channel 2/Status/Ready
//     Drive/Inputs/In/nState1 <-> DCM Status Channel 2/Status/Ready to enable
//     Drive/Inputs/In/nState1 @bit 6 <-> DCM Status Channel 2/Status/Torque reduced
//     Drive/Inputs/In/nState1 @bit 2 <-> DCM Status Channel 2/Status/Warning
//     Drive/Inputs/In/nState2 @bit 3 <-> DCM Status Channel 2/Status/Digital input 1
//     Drive/Inputs/In/nState2 @bit 4 <-> DCM Status Channel 2/Status/Digital input 2
//     Drive/Inputs/In/nState4 @bit 1 <-> WcState/InputToggle
//     Drive/Inputs/In/nState4 <-> WcState/WcState
//     Drive/Outputs/Out/nCtrl1 <-> DCM Control Channel 2/Control/Enable
//     Drive/Outputs/Out/nCtrl1 @bit 2 <-> DCM Control Channel 2/Control/Reduce torque
//     Drive/Outputs/Out/nCtrl1 @bit 1 <-> DCM Control Channel 2/Control/Reset
//     Drive/Outputs/Out/nDataOut2[0] <-> DCM Velocity Channel 2/Velocity
//     Enc/Inputs/In/nDataIn1[0] <-> ENC Status compact Channel 2/Counter value
//     Enc/Inputs/In/nDataIn2[0] <-> ENC Status compact Channel 2/Latch value
//     Enc/Inputs/In/nState1 @bit 4 <-> ENC Status compact Channel 2/Status/Counter overflow
//     Enc/Inputs/In/nState1 @bit 3 <-> ENC Status compact Channel 2/Status/Counter underflow
//     Enc/Inputs/In/nState1 @bit 7 <-> ENC Status compact Channel 2/Status/Extrapolation stall
//     Enc/Inputs/In/nState1 @bit 1 <-> ENC Status compact Channel 2/Status/Latch extern valid
//     Enc/Inputs/In/nState1 @bit 2 <-> ENC Status compact Channel 2/Status/Set counter done
//     Enc/Inputs/In/nState2 @bit 4 <-> ENC Status compact Channel 2/Status/Status of extern latch
//     Enc/Inputs/In/nState2 <-> ENC Status compact Channel 2/Status/Status of input A
//     Enc/Inputs/In/nState2 @bit 1 <-> ENC Status compact Channel 2/Status/Status of input B
//     Enc/Inputs/In/nState4 @bit 1 <-> WcState/InputToggle
//     Enc/Inputs/In/nState4 <-> WcState/WcState
//     Enc/Outputs/Out/nCtrl1 @bit 3 <-> ENC Control compact Channel 2/Control/Enable latch extern on negative edge
//     Enc/Outputs/Out/nCtrl1 @bit 1 <-> ENC Control compact Channel 2/Control/Enable latch extern on positive edge
//     Enc/Outputs/Out/nCtrl1 @bit 2 <-> ENC Control compact Channel 2/Control/Set counter
//     Enc/Outputs/Out/nDataOut1[0] <-> ENC Control compact Channel 2/Set counter value
//   NC-Task 1 SAF/Axes/NGP3 <-> Device 1 (EtherCAT)/Term 7 (EK1101)/Term 14 (EK1122)/Term 15 (EK1101)/NGP3 - NGP4 (N6) (EL7342)
//     Drive/Inputs/In/nState1 @bit 3 <-> DCM Status Channel 1/Status/Error
//     Drive/Inputs/In/nState1 @bit 5 <-> DCM Status Channel 1/Status/Moving negative
//     Drive/Inputs/In/nState1 @bit 4 <-> DCM Status Channel 1/Status/Moving positive
//     Drive/Inputs/In/nState1 @bit 1 <-> DCM Status Channel 1/Status/Ready
//     Drive/Inputs/In/nState1 <-> DCM Status Channel 1/Status/Ready to enable
//     Drive/Inputs/In/nState1 @bit 6 <-> DCM Status Channel 1/Status/Torque reduced
//     Drive/Inputs/In/nState1 @bit 2 <-> DCM Status Channel 1/Status/Warning
//     Drive/Inputs/In/nState2 @bit 3 <-> DCM Status Channel 1/Status/Digital input 1
//     Drive/Inputs/In/nState2 @bit 4 <-> DCM Status Channel 1/Status/Digital input 2
//     Drive/Inputs/In/nState2 @bit 5 <-> DCM Status Channel 1/Status/Sync error
//     Drive/Inputs/In/nState2 @bit 7 <-> DCM Status Channel 1/Status/TxPDO Toggle
//     Drive/Inputs/In/nState4 @bit 1 <-> WcState/InputToggle
//     Drive/Inputs/In/nState4 <-> WcState/WcState
//     Drive/Outputs/Out/nCtrl1 <-> DCM Control Channel 1/Control/Enable
//     Drive/Outputs/Out/nCtrl1 @bit 2 <-> DCM Control Channel 1/Control/Reduce torque
//     Drive/Outputs/Out/nCtrl1 @bit 1 <-> DCM Control Channel 1/Control/Reset
//     Drive/Outputs/Out/nCtrl1 @bit 3 <-> DCM Control Channel 1/Control/Threshold active
//     Drive/Outputs/Out/nDataOut2[0] <-> DCM Velocity Channel 1/Velocity
//     Enc/Inputs/In/nDataIn1[0] <-> ENC Status compact Channel 1/Counter value
//     Enc/Inputs/In/nDataIn2[0] <-> ENC Status compact Channel 1/Latch value
//     Enc/Inputs/In/nState1 @bit 4 <-> ENC Status compact Channel 1/Status/Counter overflow
//     Enc/Inputs/In/nState1 @bit 3 <-> ENC Status compact Channel 1/Status/Counter underflow
//     Enc/Inputs/In/nState1 @bit 7 <-> ENC Status compact Channel 1/Status/Extrapolation stall
//     Enc/Inputs/In/nState1 @bit 1 <-> ENC Status compact Channel 1/Status/Latch extern valid
//     Enc/Inputs/In/nState1 @bit 2 <-> ENC Status compact Channel 1/Status/Set counter done
//     Enc/Inputs/In/nState2 @bit 4 <-> ENC Status compact Channel 1/Status/Status of extern latch
//     Enc/Inputs/In/nState2 <-> ENC Status compact Channel 1/Status/Status of input A
//     Enc/Inputs/In/nState2 @bit 1 <-> ENC Status compact Channel 1/Status/Status of input B
//     Enc/Inputs/In/nState2 @bit 5 <-> ENC Status compact Channel 1/Status/Sync error
//     Enc/Inputs/In/nState2 @bit 7 <-> ENC Status compact Channel 1/Status/TxPDO Toggle
//     Enc/Inputs/In/nState4 @bit 1 <-> WcState/InputToggle
//     Enc/Inputs/In/nState4 <-> WcState/WcState
//     Enc/Outputs/Out/nCtrl1 @bit 3 <-> ENC Control compact Channel 1/Control/Enable latch extern on negative edge
//     Enc/Outputs/Out/nCtrl1 @bit 1 <-> ENC Control compact Channel 1/Control/Enable latch extern on positive edge
//     Enc/Outputs/Out/nCtrl1 @bit 2 <-> ENC Control compact Channel 1/Control/Set counter
//     Enc/Outputs/Out/nDataOut1[0] <-> ENC Control compact Channel 1/Set counter value
//   NC-Task 1 SAF/Axes/NGP4 <-> Device 1 (EtherCAT)/Term 7 (EK1101)/Term 14 (EK1122)/Term 15 (EK1101)/NGP3 - NGP4 (N6) (EL7342)
//     Drive/Inputs/In/nState1 @bit 3 <-> DCM Status Channel 2/Status/Error
//     Drive/Inputs/In/nState1 @bit 5 <-> DCM Status Channel 2/Status/Moving negative
//     Drive/Inputs/In/nState1 @bit 4 <-> DCM Status Channel 2/Status/Moving positive
//     Drive/Inputs/In/nState1 @bit 1 <-> DCM Status Channel 2/Status/Ready
//     Drive/Inputs/In/nState1 <-> DCM Status Channel 2/Status/Ready to enable
//     Drive/Inputs/In/nState1 @bit 6 <-> DCM Status Channel 2/Status/Torque reduced
//     Drive/Inputs/In/nState1 @bit 2 <-> DCM Status Channel 2/Status/Warning
//     Drive/Inputs/In/nState2 @bit 3 <-> DCM Status Channel 2/Status/Digital input 1
//     Drive/Inputs/In/nState2 @bit 4 <-> DCM Status Channel 2/Status/Digital input 2
//     Drive/Inputs/In/nState2 @bit 5 <-> DCM Status Channel 2/Status/Sync error
//     Drive/Inputs/In/nState2 @bit 7 <-> DCM Status Channel 2/Status/TxPDO Toggle
//     Drive/Inputs/In/nState4 @bit 1 <-> WcState/InputToggle
//     Drive/Inputs/In/nState4 <-> WcState/WcState
//     Drive/Outputs/Out/nCtrl1 <-> DCM Control Channel 2/Control/Enable
//     Drive/Outputs/Out/nCtrl1 @bit 2 <-> DCM Control Channel 2/Control/Reduce torque
//     Drive/Outputs/Out/nCtrl1 @bit 1 <-> DCM Control Channel 2/Control/Reset
//     Drive/Outputs/Out/nCtrl1 @bit 3 <-> DCM Control Channel 2/Control/Threshold active
//     Drive/Outputs/Out/nDataOut2[0] <-> DCM Velocity Channel 2/Velocity
//     Enc/Inputs/In/nDataIn1[0] <-> ENC Status compact Channel 2/Counter value
//     Enc/Inputs/In/nDataIn2[0] <-> ENC Status compact Channel 2/Latch value
//     Enc/Inputs/In/nState1 @bit 4 <-> ENC Status compact Channel 2/Status/Counter overflow
//     Enc/Inputs/In/nState1 @bit 3 <-> ENC Status compact Channel 2/Status/Counter underflow
//     Enc/Inputs/In/nState1 @bit 7 <-> ENC Status compact Channel 2/Status/Extrapolation stall
//     Enc/Inputs/In/nState1 @bit 1 <-> ENC Status compact Channel 2/Status/Latch extern valid
//     Enc/Inputs/In/nState1 @bit 2 <-> ENC Status compact Channel 2/Status/Set counter done
//     Enc/Inputs/In/nState2 @bit 4 <-> ENC Status compact Channel 2/Status/Status of extern latch
//     Enc/Inputs/In/nState2 <-> ENC Status compact Channel 2/Status/Status of input A
//     Enc/Inputs/In/nState2 @bit 1 <-> ENC Status compact Channel 2/Status/Status of input B
//     Enc/Inputs/In/nState2 @bit 5 <-> ENC Status compact Channel 2/Status/Sync error
//     Enc/Inputs/In/nState2 @bit 7 <-> ENC Status compact Channel 2/Status/TxPDO Toggle
//     Enc/Inputs/In/nState4 @bit 1 <-> WcState/InputToggle
//     Enc/Inputs/In/nState4 <-> WcState/WcState
//     Enc/Outputs/Out/nCtrl1 @bit 3 <-> ENC Control compact Channel 2/Control/Enable latch extern on negative edge
//     Enc/Outputs/Out/nCtrl1 @bit 1 <-> ENC Control compact Channel 2/Control/Enable latch extern on positive edge
//     Enc/Outputs/Out/nCtrl1 @bit 2 <-> ENC Control compact Channel 2/Control/Set counter
//     Enc/Outputs/Out/nDataOut1[0] <-> ENC Control compact Channel 2/Set counter value
//   NC-Task 1 SAF/Axes/NPC1 <-> Device 1 (EtherCAT)/Term 7 (EK1101)/Term 14 (EK1122)/Term 15 (EK1101)/NPC1 - NPC2 (N11) (EL7342)
//     Drive/Inputs/In/nState1 @bit 3 <-> DCM Status Channel 1/Status/Error
//     Drive/Inputs/In/nState1 @bit 5 <-> DCM Status Channel 1/Status/Moving negative
//     Drive/Inputs/In/nState1 @bit 4 <-> DCM Status Channel 1/Status/Moving positive
//     Drive/Inputs/In/nState1 @bit 1 <-> DCM Status Channel 1/Status/Ready
//     Drive/Inputs/In/nState1 <-> DCM Status Channel 1/Status/Ready to enable
//     Drive/Inputs/In/nState1 @bit 6 <-> DCM Status Channel 1/Status/Torque reduced
//     Drive/Inputs/In/nState1 @bit 2 <-> DCM Status Channel 1/Status/Warning
//     Drive/Inputs/In/nState2 @bit 3 <-> DCM Status Channel 1/Status/Digital input 1
//     Drive/Inputs/In/nState2 @bit 4 <-> DCM Status Channel 1/Status/Digital input 2
//     Drive/Inputs/In/nState2 @bit 5 <-> DCM Status Channel 1/Status/Sync error
//     Drive/Inputs/In/nState2 @bit 7 <-> DCM Status Channel 1/Status/TxPDO Toggle
//     Drive/Inputs/In/nState4 @bit 1 <-> WcState/InputToggle
//     Drive/Inputs/In/nState4 <-> WcState/WcState
//     Drive/Outputs/Out/nCtrl1 <-> DCM Control Channel 1/Control/Enable
//     Drive/Outputs/Out/nCtrl1 @bit 2 <-> DCM Control Channel 1/Control/Reduce torque
//     Drive/Outputs/Out/nCtrl1 @bit 1 <-> DCM Control Channel 1/Control/Reset
//     Drive/Outputs/Out/nCtrl1 @bit 3 <-> DCM Control Channel 1/Control/Threshold active
//     Drive/Outputs/Out/nDataOut2[0] <-> DCM Velocity Channel 1/Velocity
//     Enc/Inputs/In/nDataIn1[0] <-> ENC Status compact Channel 1/Counter value
//     Enc/Inputs/In/nDataIn2[0] <-> ENC Status compact Channel 1/Latch value
//     Enc/Inputs/In/nState1 @bit 4 <-> ENC Status compact Channel 1/Status/Counter overflow
//     Enc/Inputs/In/nState1 @bit 3 <-> ENC Status compact Channel 1/Status/Counter underflow
//     Enc/Inputs/In/nState1 @bit 7 <-> ENC Status compact Channel 1/Status/Extrapolation stall
//     Enc/Inputs/In/nState1 @bit 1 <-> ENC Status compact Channel 1/Status/Latch extern valid
//     Enc/Inputs/In/nState1 @bit 2 <-> ENC Status compact Channel 1/Status/Set counter done
//     Enc/Inputs/In/nState2 @bit 4 <-> ENC Status compact Channel 1/Status/Status of extern latch
//     Enc/Inputs/In/nState2 <-> ENC Status compact Channel 1/Status/Status of input A
//     Enc/Inputs/In/nState2 @bit 1 <-> ENC Status compact Channel 1/Status/Status of input B
//     Enc/Inputs/In/nState2 @bit 5 <-> ENC Status compact Channel 1/Status/Sync error
//     Enc/Inputs/In/nState2 @bit 7 <-> ENC Status compact Channel 1/Status/TxPDO Toggle
//     Enc/Inputs/In/nState4 @bit 1 <-> WcState/InputToggle
//     Enc/Inputs/In/nState4 <-> WcState/WcState
//     Enc/Outputs/Out/nCtrl1 @bit 3 <-> ENC Control compact Channel 1/Control/Enable latch extern on negative edge
//     Enc/Outputs/Out/nCtrl1 @bit 1 <-> ENC Control compact Channel 1/Control/Enable latch extern on positive edge
//     Enc/Outputs/Out/nCtrl1 @bit 2 <-> ENC Control compact Channel 1/Control/Set counter
//     Enc/Outputs/Out/nDataOut1[0] <-> ENC Control compact Channel 1/Set counter value
//   NC-Task 1 SAF/Axes/NPC2 <-> Device 1 (EtherCAT)/Term 7 (EK1101)/Term 14 (EK1122)/Term 15 (EK1101)/NPC1 - NPC2 (N11) (EL7342)
//     Drive/Inputs/In/nState1 @bit 3 <-> DCM Status Channel 2/Status/Error
//     Drive/Inputs/In/nState1 @bit 5 <-> DCM Status Channel 2/Status/Moving negative
//     Drive/Inputs/In/nState1 @bit 4 <-> DCM Status Channel 2/Status/Moving positive
//     Drive/Inputs/In/nState1 @bit 1 <-> DCM Status Channel 2/Status/Ready
//     Drive/Inputs/In/nState1 <-> DCM Status Channel 2/Status/Ready to enable
//     Drive/Inputs/In/nState1 @bit 6 <-> DCM Status Channel 2/Status/Torque reduced
//     Drive/Inputs/In/nState1 @bit 2 <-> DCM Status Channel 2/Status/Warning
//     Drive/Inputs/In/nState2 @bit 3 <-> DCM Status Channel 2/Status/Digital input 1
//     Drive/Inputs/In/nState2 @bit 4 <-> DCM Status Channel 2/Status/Digital input 2
//     Drive/Inputs/In/nState2 @bit 5 <-> DCM Status Channel 2/Status/Sync error
//     Drive/Inputs/In/nState2 @bit 7 <-> DCM Status Channel 2/Status/TxPDO Toggle
//     Drive/Inputs/In/nState4 @bit 1 <-> WcState/InputToggle
//     Drive/Inputs/In/nState4 <-> WcState/WcState
//     Drive/Outputs/Out/nCtrl1 <-> DCM Control Channel 2/Control/Enable
//     Drive/Outputs/Out/nCtrl1 @bit 2 <-> DCM Control Channel 2/Control/Reduce torque
//     Drive/Outputs/Out/nCtrl1 @bit 1 <-> DCM Control Channel 2/Control/Reset
//     Drive/Outputs/Out/nCtrl1 @bit 3 <-> DCM Control Channel 2/Control/Threshold active
//     Drive/Outputs/Out/nDataOut2[0] <-> DCM Velocity Channel 2/Velocity
//     Enc/Inputs/In/nDataIn1[0] <-> ENC Status compact Channel 2/Counter value
//     Enc/Inputs/In/nDataIn2[0] <-> ENC Status compact Channel 2/Latch value
//     Enc/Inputs/In/nState1 @bit 4 <-> ENC Status compact Channel 2/Status/Counter overflow
//     Enc/Inputs/In/nState1 @bit 3 <-> ENC Status compact Channel 2/Status/Counter underflow
//     Enc/Inputs/In/nState1 @bit 7 <-> ENC Status compact Channel 2/Status/Extrapolation stall
//     Enc/Inputs/In/nState1 @bit 1 <-> ENC Status compact Channel 2/Status/Latch extern valid
//     Enc/Inputs/In/nState1 @bit 2 <-> ENC Status compact Channel 2/Status/Set counter done
//     Enc/Inputs/In/nState2 @bit 4 <-> ENC Status compact Channel 2/Status/Status of extern latch
//     Enc/Inputs/In/nState2 <-> ENC Status compact Channel 2/Status/Status of input A
//     Enc/Inputs/In/nState2 @bit 1 <-> ENC Status compact Channel 2/Status/Status of input B
//     Enc/Inputs/In/nState2 @bit 5 <-> ENC Status compact Channel 2/Status/Sync error
//     Enc/Inputs/In/nState2 @bit 7 <-> ENC Status compact Channel 2/Status/TxPDO Toggle
//     Enc/Inputs/In/nState4 @bit 1 <-> WcState/InputToggle
//     Enc/Inputs/In/nState4 <-> WcState/WcState
//     Enc/Outputs/Out/nCtrl1 @bit 3 <-> ENC Control compact Channel 2/Control/Enable latch extern on negative edge
//     Enc/Outputs/Out/nCtrl1 @bit 1 <-> ENC Control compact Channel 2/Control/Enable latch extern on positive edge
//     Enc/Outputs/Out/nCtrl1 @bit 2 <-> ENC Control compact Channel 2/Control/Set counter
//     Enc/Outputs/Out/nDataOut1[0] <-> ENC Control compact Channel 2/Set counter value
//   NC-Task 1 SAF/Axes/NPC3 <-> Device 1 (EtherCAT)/Term 7 (EK1101)/Term 14 (EK1122)/Term 15 (EK1101)/NPC3 - NPC4 (N12) (EL7342)
//     Drive/Inputs/In/nState1 @bit 3 <-> DCM Status Channel 1/Status/Error
//     Drive/Inputs/In/nState1 @bit 5 <-> DCM Status Channel 1/Status/Moving negative
//     Drive/Inputs/In/nState1 @bit 4 <-> DCM Status Channel 1/Status/Moving positive
//     Drive/Inputs/In/nState1 @bit 1 <-> DCM Status Channel 1/Status/Ready
//     Drive/Inputs/In/nState1 <-> DCM Status Channel 1/Status/Ready to enable
//     Drive/Inputs/In/nState1 @bit 6 <-> DCM Status Channel 1/Status/Torque reduced
//     Drive/Inputs/In/nState1 @bit 2 <-> DCM Status Channel 1/Status/Warning
//     Drive/Inputs/In/nState2 @bit 3 <-> DCM Status Channel 1/Status/Digital input 1
//     Drive/Inputs/In/nState2 @bit 4 <-> DCM Status Channel 1/Status/Digital input 2
//     Drive/Inputs/In/nState2 @bit 5 <-> DCM Status Channel 1/Status/Sync error
//     Drive/Inputs/In/nState2 @bit 7 <-> DCM Status Channel 1/Status/TxPDO Toggle
//     Drive/Inputs/In/nState4 @bit 1 <-> WcState/InputToggle
//     Drive/Inputs/In/nState4 <-> WcState/WcState
//     Drive/Outputs/Out/nCtrl1 <-> DCM Control Channel 1/Control/Enable
//     Drive/Outputs/Out/nCtrl1 @bit 2 <-> DCM Control Channel 1/Control/Reduce torque
//     Drive/Outputs/Out/nCtrl1 @bit 1 <-> DCM Control Channel 1/Control/Reset
//     Drive/Outputs/Out/nCtrl1 @bit 3 <-> DCM Control Channel 1/Control/Threshold active
//     Drive/Outputs/Out/nDataOut2[0] <-> DCM Velocity Channel 1/Velocity
//     Enc/Inputs/In/nDataIn1[0] <-> ENC Status compact Channel 1/Counter value
//     Enc/Inputs/In/nDataIn2[0] <-> ENC Status compact Channel 1/Latch value
//     Enc/Inputs/In/nState1 @bit 4 <-> ENC Status compact Channel 1/Status/Counter overflow
//     Enc/Inputs/In/nState1 @bit 3 <-> ENC Status compact Channel 1/Status/Counter underflow
//     Enc/Inputs/In/nState1 @bit 7 <-> ENC Status compact Channel 1/Status/Extrapolation stall
//     Enc/Inputs/In/nState1 @bit 1 <-> ENC Status compact Channel 1/Status/Latch extern valid
//     Enc/Inputs/In/nState1 @bit 2 <-> ENC Status compact Channel 1/Status/Set counter done
//     Enc/Inputs/In/nState2 @bit 4 <-> ENC Status compact Channel 1/Status/Status of extern latch
//     Enc/Inputs/In/nState2 <-> ENC Status compact Channel 1/Status/Status of input A
//     Enc/Inputs/In/nState2 @bit 1 <-> ENC Status compact Channel 1/Status/Status of input B
//     Enc/Inputs/In/nState2 @bit 5 <-> ENC Status compact Channel 1/Status/Sync error
//     Enc/Inputs/In/nState2 @bit 7 <-> ENC Status compact Channel 1/Status/TxPDO Toggle
//     Enc/Inputs/In/nState4 @bit 1 <-> WcState/InputToggle
//     Enc/Inputs/In/nState4 <-> WcState/WcState
//     Enc/Outputs/Out/nCtrl1 @bit 3 <-> ENC Control compact Channel 1/Control/Enable latch extern on negative edge
//     Enc/Outputs/Out/nCtrl1 @bit 1 <-> ENC Control compact Channel 1/Control/Enable latch extern on positive edge
//     Enc/Outputs/Out/nCtrl1 @bit 2 <-> ENC Control compact Channel 1/Control/Set counter
//     Enc/Outputs/Out/nDataOut1[0] <-> ENC Control compact Channel 1/Set counter value
//   NC-Task 1 SAF/Axes/NPC4 <-> Device 1 (EtherCAT)/Term 7 (EK1101)/Term 14 (EK1122)/Term 15 (EK1101)/NPC3 - NPC4 (N12) (EL7342)
//     Drive/Inputs/In/nState1 @bit 3 <-> DCM Status Channel 2/Status/Error
//     Drive/Inputs/In/nState1 @bit 5 <-> DCM Status Channel 2/Status/Moving negative
//     Drive/Inputs/In/nState1 @bit 4 <-> DCM Status Channel 2/Status/Moving positive
//     Drive/Inputs/In/nState1 @bit 1 <-> DCM Status Channel 2/Status/Ready
//     Drive/Inputs/In/nState1 <-> DCM Status Channel 2/Status/Ready to enable
//     Drive/Inputs/In/nState1 @bit 6 <-> DCM Status Channel 2/Status/Torque reduced
//     Drive/Inputs/In/nState1 @bit 2 <-> DCM Status Channel 2/Status/Warning
//     Drive/Inputs/In/nState2 @bit 3 <-> DCM Status Channel 2/Status/Digital input 1
//     Drive/Inputs/In/nState2 @bit 4 <-> DCM Status Channel 2/Status/Digital input 2
//     Drive/Inputs/In/nState2 @bit 5 <-> DCM Status Channel 2/Status/Sync error
//     Drive/Inputs/In/nState2 @bit 7 <-> DCM Status Channel 2/Status/TxPDO Toggle
//     Drive/Inputs/In/nState4 @bit 1 <-> WcState/InputToggle
//     Drive/Inputs/In/nState4 <-> WcState/WcState
//     Drive/Outputs/Out/nCtrl1 <-> DCM Control Channel 2/Control/Enable
//     Drive/Outputs/Out/nCtrl1 @bit 2 <-> DCM Control Channel 2/Control/Reduce torque
//     Drive/Outputs/Out/nCtrl1 @bit 1 <-> DCM Control Channel 2/Control/Reset
//     Drive/Outputs/Out/nCtrl1 @bit 3 <-> DCM Control Channel 2/Control/Threshold active
//     Drive/Outputs/Out/nDataOut2[0] <-> DCM Velocity Channel 2/Velocity
//     Enc/Inputs/In/nDataIn1[0] <-> ENC Status compact Channel 2/Counter value
//     Enc/Inputs/In/nDataIn2[0] <-> ENC Status compact Channel 2/Latch value
//     Enc/Inputs/In/nState1 @bit 4 <-> ENC Status compact Channel 2/Status/Counter overflow
//     Enc/Inputs/In/nState1 @bit 3 <-> ENC Status compact Channel 2/Status/Counter underflow
//     Enc/Inputs/In/nState1 @bit 7 <-> ENC Status compact Channel 2/Status/Extrapolation stall
//     Enc/Inputs/In/nState1 @bit 1 <-> ENC Status compact Channel 2/Status/Latch extern valid
//     Enc/Inputs/In/nState1 @bit 2 <-> ENC Status compact Channel 2/Status/Set counter done
//     Enc/Inputs/In/nState2 @bit 4 <-> ENC Status compact Channel 2/Status/Status of extern latch
//     Enc/Inputs/In/nState2 <-> ENC Status compact Channel 2/Status/Status of input A
//     Enc/Inputs/In/nState2 @bit 1 <-> ENC Status compact Channel 2/Status/Status of input B
//     Enc/Inputs/In/nState2 @bit 5 <-> ENC Status compact Channel 2/Status/Sync error
//     Enc/Inputs/In/nState2 @bit 7 <-> ENC Status compact Channel 2/Status/TxPDO Toggle
//     Enc/Inputs/In/nState4 @bit 1 <-> WcState/InputToggle
//     Enc/Inputs/In/nState4 <-> WcState/WcState
//     Enc/Outputs/Out/nCtrl1 @bit 3 <-> ENC Control compact Channel 2/Control/Enable latch extern on negative edge
//     Enc/Outputs/Out/nCtrl1 @bit 1 <-> ENC Control compact Channel 2/Control/Enable latch extern on positive edge
//     Enc/Outputs/Out/nCtrl1 @bit 2 <-> ENC Control compact Channel 2/Control/Set counter
//     Enc/Outputs/Out/nDataOut1[0] <-> ENC Control compact Channel 2/Set counter value
//   NC-Task 1 SAF/Axes/NSH1 <-> Device 1 (EtherCAT)/Term 7 (EK1101)/Term 14 (EK1122)/Term 15 (EK1101)/NSH1 (N16) (EL7047)
//     Drive/Inputs/In/nState1 @bit 3 <-> STM Status/Status/Error
//     Drive/Inputs/In/nState1 @bit 7 <-> STM Status/Status/Motor stall
//     Drive/Inputs/In/nState1 @bit 5 <-> STM Status/Status/Moving negative
//     Drive/Inputs/In/nState1 @bit 4 <-> STM Status/Status/Moving positive
//     Drive/Inputs/In/nState1 @bit 1 <-> STM Status/Status/Ready
//     Drive/Inputs/In/nState1 <-> STM Status/Status/Ready to enable
//     Drive/Inputs/In/nState1 @bit 6 <-> STM Status/Status/Torque reduced
//     Drive/Inputs/In/nState1 @bit 2 <-> STM Status/Status/Warning
//     Drive/Inputs/In/nState2 @bit 3 <-> STM Status/Status/Digital input 1
//     Drive/Inputs/In/nState2 @bit 4 <-> STM Status/Status/Digital input 2
//     Drive/Inputs/In/nState2 @bit 5 <-> STM Status/Status/Sync error
//     Drive/Inputs/In/nState2 @bit 7 <-> STM Status/Status/TxPDO Toggle
//     Drive/Inputs/In/nState4 @bit 1 <-> WcState/InputToggle
//     Drive/Inputs/In/nState4 <-> WcState/WcState
//     Drive/Outputs/Out/nCtrl1 <-> STM Control/Control/Enable
//     Drive/Outputs/Out/nCtrl1 @bit 2 <-> STM Control/Control/Reduce torque
//     Drive/Outputs/Out/nCtrl1 @bit 1 <-> STM Control/Control/Reset
//     Drive/Outputs/Out/nCtrl2 @bit 3 <-> STM Control/Control/Digital output 1
//     Drive/Outputs/Out/nDataOut2[0] <-> STM Velocity/Velocity
//     Enc/Inputs/In/nDataIn1[0] <-> ENC Status compact/Counter value
//     Enc/Inputs/In/nDataIn2[0] <-> ENC Status compact/Latch value
//     Enc/Inputs/In/nState1 @bit 4 <-> ENC Status compact/Status/Counter overflow
//     Enc/Inputs/In/nState1 @bit 3 <-> ENC Status compact/Status/Counter underflow
//     Enc/Inputs/In/nState1 @bit 7 <-> ENC Status compact/Status/Extrapolation stall
//     Enc/Inputs/In/nState1 <-> ENC Status compact/Status/Latch C valid
//     Enc/Inputs/In/nState1 @bit 1 <-> ENC Status compact/Status/Latch extern valid
//     Enc/Inputs/In/nState1 @bit 2 <-> ENC Status compact/Status/Set counter done
//     Enc/Inputs/In/nState2 @bit 4 <-> ENC Status compact/Status/Status of extern latch
//     Enc/Inputs/In/nState2 <-> ENC Status compact/Status/Status of input A
//     Enc/Inputs/In/nState2 @bit 1 <-> ENC Status compact/Status/Status of input B
//     Enc/Inputs/In/nState2 @bit 2 <-> ENC Status compact/Status/Status of input C
//     Enc/Inputs/In/nState2 @bit 5 <-> ENC Status compact/Status/Sync error
//     Enc/Inputs/In/nState2 @bit 7 <-> ENC Status compact/Status/TxPDO Toggle
//     Enc/Inputs/In/nState4 @bit 1 <-> WcState/InputToggle
//     Enc/Inputs/In/nState4 <-> WcState/WcState
//     Enc/Outputs/Out/nCtrl1 <-> ENC Control compact/Control/Enable latch C
//     Enc/Outputs/Out/nCtrl1 @bit 3 <-> ENC Control compact/Control/Enable latch extern on negative edge
//     Enc/Outputs/Out/nCtrl1 @bit 1 <-> ENC Control compact/Control/Enable latch extern on positive edge
//     Enc/Outputs/Out/nCtrl1 @bit 2 <-> ENC Control compact/Control/Set counter
//     Enc/Outputs/Out/nDataOut1[0] <-> ENC Control compact/Set counter value
//   NC-Task 1 SAF/Axes/NSH2 <-> Device 1 (EtherCAT)/Term 7 (EK1101)/Term 14 (EK1122)/Term 15 (EK1101)/NSH2 (N17) (EL7047)
//     Drive/Inputs/In/nState1 @bit 3 <-> STM Status/Status/Error
//     Drive/Inputs/In/nState1 @bit 7 <-> STM Status/Status/Motor stall
//     Drive/Inputs/In/nState1 @bit 5 <-> STM Status/Status/Moving negative
//     Drive/Inputs/In/nState1 @bit 4 <-> STM Status/Status/Moving positive
//     Drive/Inputs/In/nState1 @bit 1 <-> STM Status/Status/Ready
//     Drive/Inputs/In/nState1 <-> STM Status/Status/Ready to enable
//     Drive/Inputs/In/nState1 @bit 6 <-> STM Status/Status/Torque reduced
//     Drive/Inputs/In/nState1 @bit 2 <-> STM Status/Status/Warning
//     Drive/Inputs/In/nState2 @bit 3 <-> STM Status/Status/Digital input 1
//     Drive/Inputs/In/nState2 @bit 4 <-> STM Status/Status/Digital input 2
//     Drive/Inputs/In/nState2 @bit 5 <-> STM Status/Status/Sync error
//     Drive/Inputs/In/nState2 @bit 7 <-> STM Status/Status/TxPDO Toggle
//     Drive/Inputs/In/nState4 @bit 1 <-> WcState/InputToggle
//     Drive/Inputs/In/nState4 <-> WcState/WcState
//     Drive/Outputs/Out/nCtrl1 <-> STM Control/Control/Enable
//     Drive/Outputs/Out/nCtrl1 @bit 2 <-> STM Control/Control/Reduce torque
//     Drive/Outputs/Out/nCtrl1 @bit 1 <-> STM Control/Control/Reset
//     Drive/Outputs/Out/nCtrl2 @bit 3 <-> STM Control/Control/Digital output 1
//     Drive/Outputs/Out/nDataOut2[0] <-> STM Velocity/Velocity
//     Enc/Inputs/In/nDataIn1[0] <-> ENC Status compact/Counter value
//     Enc/Inputs/In/nDataIn2[0] <-> ENC Status compact/Latch value
//     Enc/Inputs/In/nState1 @bit 4 <-> ENC Status compact/Status/Counter overflow
//     Enc/Inputs/In/nState1 @bit 3 <-> ENC Status compact/Status/Counter underflow
//     Enc/Inputs/In/nState1 @bit 7 <-> ENC Status compact/Status/Extrapolation stall
//     Enc/Inputs/In/nState1 <-> ENC Status compact/Status/Latch C valid
//     Enc/Inputs/In/nState1 @bit 1 <-> ENC Status compact/Status/Latch extern valid
//     Enc/Inputs/In/nState1 @bit 2 <-> ENC Status compact/Status/Set counter done
//     Enc/Inputs/In/nState2 @bit 4 <-> ENC Status compact/Status/Status of extern latch
//     Enc/Inputs/In/nState2 <-> ENC Status compact/Status/Status of input A
//     Enc/Inputs/In/nState2 @bit 1 <-> ENC Status compact/Status/Status of input B
//     Enc/Inputs/In/nState2 @bit 2 <-> ENC Status compact/Status/Status of input C
//     Enc/Inputs/In/nState2 @bit 5 <-> ENC Status compact/Status/Sync error
//     Enc/Inputs/In/nState2 @bit 7 <-> ENC Status compact/Status/TxPDO Toggle
//     Enc/Inputs/In/nState4 @bit 1 <-> WcState/InputToggle
//     Enc/Inputs/In/nState4 <-> WcState/WcState
//     Enc/Outputs/Out/nCtrl1 <-> ENC Control compact/Control/Enable latch C
//     Enc/Outputs/Out/nCtrl1 @bit 3 <-> ENC Control compact/Control/Enable latch extern on negative edge
//     Enc/Outputs/Out/nCtrl1 @bit 1 <-> ENC Control compact/Control/Enable latch extern on positive edge
//     Enc/Outputs/Out/nCtrl1 @bit 2 <-> ENC Control compact/Control/Set counter
//     Enc/Outputs/Out/nDataOut1[0] <-> ENC Control compact/Set counter value
//   NC-Task 1 SAF/Axes/NSH3 <-> Device 1 (EtherCAT)/Term 7 (EK1101)/Term 14 (EK1122)/Term 15 (EK1101)/NSH3 (N18) (EL7047)
//     Drive/Inputs/In/nState1 @bit 3 <-> STM Status/Status/Error
//     Drive/Inputs/In/nState1 @bit 7 <-> STM Status/Status/Motor stall
//     Drive/Inputs/In/nState1 @bit 5 <-> STM Status/Status/Moving negative
//     Drive/Inputs/In/nState1 @bit 4 <-> STM Status/Status/Moving positive
//     Drive/Inputs/In/nState1 @bit 1 <-> STM Status/Status/Ready
//     Drive/Inputs/In/nState1 <-> STM Status/Status/Ready to enable
//     Drive/Inputs/In/nState1 @bit 6 <-> STM Status/Status/Torque reduced
//     Drive/Inputs/In/nState1 @bit 2 <-> STM Status/Status/Warning
//     Drive/Inputs/In/nState2 @bit 3 <-> STM Status/Status/Digital input 1
//     Drive/Inputs/In/nState2 @bit 4 <-> STM Status/Status/Digital input 2
//     Drive/Inputs/In/nState2 @bit 5 <-> STM Status/Status/Sync error
//     Drive/Inputs/In/nState2 @bit 7 <-> STM Status/Status/TxPDO Toggle
//     Drive/Inputs/In/nState4 @bit 1 <-> WcState/InputToggle
//     Drive/Inputs/In/nState4 <-> WcState/WcState
//     Drive/Outputs/Out/nCtrl1 <-> STM Control/Control/Enable
//     Drive/Outputs/Out/nCtrl1 @bit 2 <-> STM Control/Control/Reduce torque
//     Drive/Outputs/Out/nCtrl1 @bit 1 <-> STM Control/Control/Reset
//     Drive/Outputs/Out/nCtrl2 @bit 3 <-> STM Control/Control/Digital output 1
//     Drive/Outputs/Out/nDataOut2[0] <-> STM Velocity/Velocity
//     Enc/Inputs/In/nDataIn1[0] <-> ENC Status compact/Counter value
//     Enc/Inputs/In/nDataIn2[0] <-> ENC Status compact/Latch value
